# B&R Automation Studio project Soiled_PLC (part 17)

#### Main.st
```iecst
PROGRAM _INIT
	state 			:= 0;
	pFileName 	:= ADR('Test');//file name
	pFileDevice	:=ADR('FTP');//Can be file name set up in AS, or Devlink folder name
	//pDevLinkParameter := ADR('/DEVICE=C:\\Projects\FTP\Test');//Path for Devlink
	pDevLinkParameter := ADR('/SIP=10.8.4.211 /PROTOCOL=ftp /USER=SUP /PASSWORD=12345');
	pMemCard	:= ADR('memcard');//Pointer to memory card file device
	pUSB 		:= ADR('USB');
	//Create temporary memory object for the files to be read into..
	sizeTempMem := 30000000; //Allocate 30MB of free memory
	TMP_alloc(sizeTempMem,ADR(pTempMem));
END_PROGRAM

PROGRAM _CYCLIC

	CASE state OF
		XML_READER_IDLE:

		XML_READER_COPY_FILE_TO_MEMCARD: //Copy File from FTP Server to Memcard.
			fileCopyFromDev.enable := 1;
			fileCopyFromDev.pFileName := pFileName;// Name of file to copy
			fileCopyFromDev.pFileDevice := pFileDevice;//Folder to copy from
			fileCopyFromDev.pDevLinkParameter := pDevLinkParameter;//Parameters for Devlink...
			fileCopyFromDev.pDest := pFileName;
			fileCopyFromDev.pDestDev := pMemCard;//pUSB;
			fileCopyFromDev();
			IF fileCopyFromDev.status = ERR_OK THEN
				state := XML_READER_DECODE_FILE;
			ELSIF fileCopyFromDev.status = 26228 THEN//ERR_DDFI_NETIO_DLINK THEN //No file available on network... use local memory card file..
				state := XML_READER_DECODE_FILE;
			ELSIF fileCopyFromDev.status <> ERR_FUB_BUSY THEN
				state := XML_READER_DECODE_ERROR;
			END_IF;

		XML_READER_DECODE_FILE:
		//Decode XML File Copy into temp memory then read...
			n:= 0;
			FOR n:= 0 TO 100 DO //Use loop to increase scan time..
				CASE xmlReader OF
					0://Copy into memory
						fiToMem.enable := 1;
						fiToMem.pFileDevice := pMemCard;
						fiToMem.pFileName := pFileName;
						fiToMem.pTempMem := pTempMem;
						fiToMem.sizeTempMem := sizeTempMem;
						fiToMem();
						IF fiToMem.status = ERR_OK THEN
							memcpy(ADR(testString),pTempMem,SIZEOF(testString));
							xmlReader := 10;
						ELSIF fiToMem.status <> ERR_FUB_BUSY THEN
							xmlReader := 100;
						END_IF;

					10://Copy data to file for test..
						fileWrite.enable := 1;
						fileWrite.mode := FILE_SAVE;
						fileWrite.Offset := 0;
						fileWrite.pData := pTempMem;
						fileWrite.sizeData := fiToMem.fiSize;//responseHeader.contentLength;
						fileWrite.pFileDevice := pUSB;
						fileWrite.pFileName := ADR('FTP_Test.xml');
						fileWrite();
						IF fileWrite.status = ERR_OK THEN
							xmlReader := 1;
						END_IF;

					1://Create XML Reaser
						xmlReadCreate.enable := 1;
						xmlReadCreate.memorySize := fiToMem.fiSize;
						xmlReadCreate.pXmlMemory := pTempMem;
						xmlReadCreate();
						IF xmlReadCreate.status = ERR_OK THEN
							lineCount := 0;
							xmlReader := 2;
						ELSIF xmlReadCreate.status <> ERR_FUB_BUSY THEN
							xmlReader := 100;
						END_IF;

					2://Search for 'Config setting'
						xmlReadNode.enable := 1;
						xmlReadNode.ident := xmlReadCreate.ident;
						xmlReadNode.forceRead := 0;
						xmlReadNode.skipSubtree := 0;
						xmlReadNode.pName := ADR(xmlName);
						xmlReadNode.nameSize := SIZEOF(xmlName);
						xmlReadNode.pValue := ADR(xmlValue);
						xmlReadNode.valueSize := SIZEOF(xmlValue);
						xmlReadNode();
						IF xmlReadNode.status = ERR_OK THEN
							IF xmlName = 'Config' THEN
								lineCount := lineCount + 1;
								xmlIndex := 0;
								xmlReader := 3;
							END_IF;
						ELSIF xmlReadNode.status = xmlERR_NO_FURTHER_XML_NODE THEN
							xmlReader := 4;//End of file
						ELSIF xmlReadNode.status <> ERR_FUB_BUSY THEN
							xmlReader := 100;
						END_IF

					3://Decode XML elements
						xmlReadAttNum.enable := 1;
						xmlReadAttNum.ident := xmlReadCreate.ident;
						xmlReadAttNum.index := xmlIndex;
						xmlReadAttNum.pName := ADR(xmlName);
						xmlReadAttNum.nameSize := SIZEOF(xmlName);
						xmlReadAttNum.pValue := ADR(xmlValue);
						xmlReadAttNum.valueSize := SIZEOF(xmlValue);
						xmlReadAttNum();
						IF xmlReadAttNum.status = ERR_OK THEN
							IF xmlName = 'Property' THEN
								xmlProperty := xmlValue;
							ELSIF xmlName = 'Index' THEN
								xmlPropertyIndex := atoi(ADR(xmlValue));
							ELSIF xmlName =	'FirstBag' THEN
								IF (xmlProperty = 'Line') AND (xmlPropertyIndex > 0) AND  (xmlPropertyIndex <= MAX_LINES) THEN
									Line[xmlPropertyIndex].FirstBag := DINT_TO_UINT(atoi(ADR(xmlValue)));
								END_IF;
							ELSIF xmlName = 'LastBag' THEN
								IF (xmlProperty = 'Line') AND (xmlPropertyIndex > 0) AND  (xmlPropertyIndex <= MAX_LINES) THEN
									Line[xmlPropertyIndex].LastBag := DINT_TO_UINT(atoi(ADR(xmlValue)));
								END_IF;
							END_IF;
							xmlIndex := xmlIndex + 1;
						ELSIF xmlReadAttNum.status = xmlERR_INVALID_ATTRIBUTE_INDEX THEN//No more elements go back to beginning..
							xmlReader := 2;
						ELSIF xmlReadAttNum.status <> ERR_FUB_BUSY THEN
							xmlReader := 100;
						END_IF

					4://Close XML Reader
						xmlCloseReader.enable := 1;
						xmlCloseReader.ident := xmlReadCreate.ident;
						xmlCloseReader();
						IF xmlCloseReader.status = ERR_OK THEN
							xmlReader := 99;
						ELSIF xmlCloseReader.status <> ERR_FUB_BUSY THEN
							xmlReader := 100;
						END_IF;

					99:
						state := 99;
						xmlReader := 0;
					100://Error
						state := 100;
						xmlReader := 0;

				END_CASE;
				IF xmlReader = 0 THEN
					EXIT;
				END_IF;
			END_FOR;

		XML_READER_DECODE_ERROR:

		ELSE
			state := XML_READER_IDLE;

	END_CASE;

END_PROGRAM
```

### Program Logical/File_System/zzXMLFileViaHttp (IEC)

#### Variables.var
```iecst
(*State Constants*)
VAR CONSTANT
	XML_READER_IDLE : UINT := 0;
	XML_READER_READ_FROM_HTTP : UINT := 1;
	XML_READER_DECODE_FILE : UINT := 2;
	XML_READER_DECODE_ERROR : UINT := 99;
END_VAR
(**Local Vars*)
VAR
	state : UINT;
	error : UINT;
	pTempMem : UDINT;
	sizeTempMem : UDINT;
	pFileName : UDINT;
	pFileDevice : UDINT;
	pDevLinkParameter : UDINT;
	pMemCard : UDINT;
	fileCopyFromDev : FileCopyFromDev;
	pUSB : UDINT;
	n : UINT;
	xmlReader : UINT;
	lineCount : UINT;
	xmlName : STRING[100];
	xmlValue : STRING[100];
	xmlIndex : UDINT;
	xmlProperty : STRING[100];
	xmlPropertyIndex : DINT;
	fiToMem : fileToMem;
	xmlReadCreate : xmlCreateMemoryReader;
	xmlReadNode : xmlReadNextNode;
	xmlReadAttNum : xmlReadAttributeNr;
	xmlCloseReader : xmlCloseMemoryReader;
	pHost : UDINT;
	URL : STRING[30];
	pResponseHeader : UDINT;
	responseHeader : httpResponseHeader_t;
	pRequestHeader : UDINT;
	requestHeader : httpRequestHeader_t;
	pStatistics : UDINT;
	Statistics : httpStatistics_t;
	pSendData : UDINT;
	sendData : STRING[100];
	pResponseData : UDINT;
	responseData : ARRAY[0..99] OF USINT;
	pUri : UDINT;
	testAbort : BOOL;
	http_Client : httpClient;
	testSend : BOOL;
	fileWrite : fileReadWrite;
	fiLength : UDINT;
END_VAR
```

#### Main.st
```iecst
PROGRAM _INIT
	pHost := ADR('10.8.4.102');
	URL := '/plctalk/api/values/3';
	pUri := ADR(URL);
	pResponseHeader := ADR(responseHeader);
	pRequestHeader := ADR(requestHeader);
	pStatistics := ADR(Statistics);
	pSendData := ADR(sendData);
	pResponseData := ADR(responseData);

	state 			:= 0;
	pFileName 	:= ADR('Test');//file name
	//pFileDevice	:=ADR('FTP');//Can be file name set up in AS, or Devlink folder name
	//pDevLinkParameter := ADR('/DEVICE=C:\\Projects\FTP\Test');//Path for Devlink
	//pDevLinkParameter := ADR('/SIP=10.8.4.211 /PROTOCOL=ftp /USER=SUP /PASSWORD=12345');
	pMemCard	:= ADR('memcard');//Pointer to memory card file device
	pUSB 		:= ADR('USB');
	//Create temporary memory object for the files to be read into..
	sizeTempMem := 10000000; //Allocate 10MB of free memory
	TMP_alloc(sizeTempMem,ADR(pTempMem));
END_PROGRAM

PROGRAM _CYCLIC
http_Client.enable := 1;
http_Client.send := testSend;
http_Client.abort := testAbort;
http_Client.option := httpOPTION_HTTP_11;
http_Client.pHost := pHost;
http_Client.hostPort := 0;//20997;
http_Client.pUri := pUri;
http_Client.pRequestHeader := 0;//pRequestHeader;
http_Client.pRequestData := pSendData;
http_Client.requestDataLen := LEN(sendData);
http_Client.pResponseHeader := pResponseHeader;
http_Client.pResponseData := pTempMem; //pResponseData;
http_Client.responseDataSize := sizeTempMem;//SIZEOF(responseData);
http_Client.pStatistics := pStatistics;
http_Client.method := httpMETHOD_GET;
http_Client();

	CASE state OF
		XML_READER_IDLE:
			testSend := 0;

		XML_READER_READ_FROM_HTTP: //Copy File from FTP Server to Memcard.
			testSend := 1;
			IF (http_Client.phase = httpPHASE_RECEIVED) THEN
				state := 10;//XML_READER_DECODE_FILE;
				IF (responseHeader.contentLength > 0) THEN
					IF (responseHeader.contentLength <= SIZEOF(responseData)) THEN
						memcpy(pResponseData,pTempMem,responseHeader.contentLength);
					ELSE
						memcpy(pResponseData,pTempMem,SIZEOF(responseData));
					END_IF;
				END_IF;
			END_IF;

		10://Copy data to file for test..
			fileWrite.enable := 1;
			fileWrite.mode := FILE_SAVE;
			fileWrite.Offset := 0;
			fileWrite.pData := pTempMem;
			fileWrite.sizeData := responseHeader.contentLength;
			fileWrite.pFileDevice := pUSB;
			fileWrite.pFileName := ADR('text.xml');
			fileWrite();
			IF fileWrite.status = ERR_OK THEN
				state := XML_READER_DECODE_FILE;
			ELSIF fileWrite.status <> ERR_FUB_BUSY THEN
				state := XML_READER_DECODE_FILE;
			END_IF;

		XML_READER_DECODE_FILE:
		//Decode XML File Copy into temp memory then read...
			n:= 0;
			FOR n:= 0 TO 100 DO //Use loop to increase scan time..
				CASE xmlReader OF
					0://Copy into memory
//						fiToMem.enable := 1;
//						fiToMem.pFileDevice := pMemCard;
//						fiToMem.pFileName := pFileName;
//						fiToMem.pTempMem := pTempMem;
//						fiToMem.sizeTempMem := sizeTempMem;
//						fiToMem();
//						IF fiToMem.status = ERR_OK THEN
							xmlReader := 1;
//						ELSIF fiToMem.status <> ERR_FUB_BUSY THEN
//							xmlReader := 100;
//						END_IF;

					1://Create XML Reaser
						xmlReadCreate.enable := 1;
						xmlReadCreate.memorySize := responseHeader.contentLength;
						xmlReadCreate.pXmlMemory := pTempMem;
						xmlReadCreate();
						IF xmlReadCreate.status = ERR_OK THEN
							lineCount := 0;
							xmlReader := 2;
						ELSIF xmlReadCreate.status <> ERR_FUB_BUSY THEN
							xmlReader := 100;
						END_IF;

					2://Search for 'Config setting'
						xmlReadNode.enable := 1;
						xmlReadNode.ident := xmlReadCreate.ident;
						xmlReadNode.forceRead := 0;
						xmlReadNode.skipSubtree := 0;
						xmlReadNode.pName := ADR(xmlName);
						xmlReadNode.nameSize := SIZEOF(xmlName);
						xmlReadNode.pValue := ADR(xmlValue);
						xmlReadNode.valueSize := SIZEOF(xmlValue);
						xmlReadNode();
						IF xmlReadNode.status = ERR_OK THEN
							IF xmlName = 'Config' THEN
								lineCount := lineCount + 1;
								xmlIndex := 0;
								xmlReader := 3;
							END_IF;
						ELSIF xmlReadNode.status = xmlERR_NO_FURTHER_XML_NODE THEN
							xmlReader := 4;//End of file
						ELSIF xmlReadNode.status <> ERR_FUB_BUSY THEN
							xmlReader := 100;
						END_IF

					3://Decode XML elements
						xmlReadAttNum.enable := 1;
						xmlReadAttNum.ident := xmlReadCreate.ident;
						xmlReadAttNum.index := xmlIndex;
						xmlReadAttNum.pName := ADR(xmlName);
						xmlReadAttNum.nameSize := SIZEOF(xmlName);
						xmlReadAttNum.pValue := ADR(xmlValue);
						xmlReadAttNum.valueSize := SIZEOF(xmlValue);
						xmlReadAttNum();
						IF xmlReadAttNum.status = ERR_OK THEN
							IF xmlName = 'Property' THEN
								xmlProperty := xmlValue;
							ELSIF xmlName = 'Index' THEN
								xmlPropertyIndex := atoi(ADR(xmlValue));
							ELSIF xmlName =	'FirstBag' THEN
								IF (xmlProperty = 'Line') AND (xmlPropertyIndex > 0) AND  (xmlPropertyIndex <= MAX_LINES) THEN
									Line[xmlPropertyIndex].FirstBag := DINT_TO_UINT(atoi(ADR(xmlValue)));
								END_IF;
							ELSIF xmlName = 'LastBag' THEN
								IF (xmlProperty = 'Line') AND (xmlPropertyIndex > 0) AND  (xmlPropertyIndex <= MAX_LINES) THEN
									Line[xmlPropertyIndex].LastBag := DINT_TO_UINT(atoi(ADR(xmlValue)));
								END_IF;
							END_IF;
							xmlIndex := xmlIndex + 1;
						ELSIF xmlReadAttNum.status = xmlERR_INVALID_ATTRIBUTE_INDEX THEN//No more elements go back to beginning..
							xmlReader := 2;
						ELSIF xmlReadAttNum.status <> ERR_FUB_BUSY THEN
							xmlReader := 100;
						END_IF

					4://Close XML Reader
						xmlCloseReader.enable := 1;
						xmlCloseReader.ident := xmlReadCreate.ident;
						xmlCloseReader();
						IF xmlCloseReader.status = ERR_OK THEN
							xmlReader := 99;
						ELSIF xmlCloseReader.status <> ERR_FUB_BUSY THEN
							xmlReader := 100;
						END_IF;

					99:
						state := 99;
						xmlReader := 0;

					100://Error
						state := 100;
						xmlReader := 0;

				END_CASE;
				IF xmlReader = 0 THEN
					//memset(pTempMem,0,sizeTempMem); //Clear memory when finish
					EXIT;
				END_IF;
			END_FOR;

		XML_READER_DECODE_ERROR:

		100://ERROR

		ELSE
			state := XML_READER_IDLE;

	END_CASE;

END_PROGRAM
```

### Program Logical/File_System/sendXML (IEC)

#### Variables.var - Local variables
```iecst
VAR
	xml : xml_typ;
	state : REFERENCE TO USINT;
	xmlWriter : xml_writer_typ;
	testData : testData_typ;
	status : UINT;
	pStructName : UDINT;
	index : UINT;
	pvName : STRING[50];
	structName : STRING[32];
	taskName : STRING[55];
	encodeXML : WriteXMLFromStructure;
	pv_dataLen : UINT;
	noOfElements : UINT;
	pvStatus : UINT;
	pv_dataType : UINT;
	pvFullName : STRING[50];
	subIndex : UINT;
	pvValue : UDINT;
	batch : test2;
	enable : BOOL;
	testTim : BOOL;
END_VAR
```

#### Types.typ - Local data types
```iecst
TYPE
	xml_typ : 	STRUCT
		Write : xml_writer_typ;
	END_STRUCT;
	xml_writer_typ : 	STRUCT
		State : USINT; (**State of the writer...*)
		Functions : xml_write_fub_typ;
	END_STRUCT;
	xml_write_fub_typ : 	STRUCT
		CreateMemWriter : xmlCreateMemoryWriter;
	END_STRUCT;
	testData_typ : 	STRUCT
		BatchID : USINT;
		ElementArray : ARRAY[0..9]OF USINT;
		Structure : test2;
	END_STRUCT;
	test2 : 	STRUCT
		StrElement : USINT;
		stElement2 : USINT;
	END_STRUCT;
END_TYPE
```

#### Main.st - Init, cyclic, exit code
```iecst
PROGRAM _INIT
	(* Insert code here *)

END_PROGRAM

PROGRAM _CYCLIC
	//_compileXML;
	DF2327SortedBatches;

	DF2327SortedBatches.updatedAt := CurrentTimestamp;
	batch;

	encodeXML.enable := enable;
	encodeXML.pStructName := ADR('DF2327SortedBatches');
	encodeXML.pData := ADR(Data);
	encodeXML.sizeData := SIZEOF(Data);
	encodeXML();
	IF (encodeXML.status = ERR_OK) THEN
		enable := 0;
	ELSIF (encodeXML.status <> ERR_FUB_BUSY) THEN

	END_IF;

	IF testTim THEN
		memcpy(ADR(Data),ADR(''),SIZEOF(Data));
		testTim := 0;
	 END_IF;
END_PROGRAM
```

#### compileXML.st
```iecst
ACTION _compileXML:
	state ACCESS ADR(xml.Write.State);
	testData;

	CASE xmlWriter.State OF

		30://Open an XML writer
			xmlWriter.Functions.CreateMemWriter.enable := 1;
			IF (xmlWriter.Functions.CreateMemWriter.status = ERR_OK) THEN
				xmlWriter.State := 1;
			END_IF;

		1:// Write the document header
			//Write the encoding version.

		10://Wait.
			structName := 'testData';
			pStructName := ADR(structName);

		11://Read the Data structure so we can manipulate into XML
			//What have to pass in the structure Name..
			// Only pass the structure name -- The code will handle it if it;s global or local
			status := PV_item(pStructName,index,ADR(pvName));
			IF (status = ERR_OK) THEN
				//Build the pvFullName
				brsstrcpy(ADR(pvFullName),ADR(structName));
				brsstrcat(ADR(pvFullName),ADR('.'));
				brsstrcat(ADR(pvFullName),ADR(pvName));
				xmlWriter.State := 20;
			ELSIF (status =  ERR_SYS_PV_NOT_FOUND) THEN
				//Add the taskname in front of the var to declare it as local.
				ST_name(0,ADR(taskName),0);
				brsstrcat(ADR(taskName),ADR(':'));
				brsstrcat(ADR(taskName),ADR(structName));
				brsstrcpy(ADR(structName),ADR(taskName));
				pStructName := ADR(structName);
			END_IF;

		20://Get the info..
			pvStatus := PV_ninfo(ADR(pvFullName),ADR(pv_dataType),ADR(pv_dataLen),ADR(noOfElements));
			IF pvStatus = ERR_OK THEN
				xmlWriter.State := 21;
			END_IF;

		21://
			//Don't use get val as it doesn;t support strings..
			//We can get the address and memcpy... then cast to string

			//pvStatus := PV_xgetval(ADR(pvFullName),subIndex,ADR(pvValue),2);
			IF pvStatus = ERR_OK THEN
				xmlWriter.State := 22;
			END_IF;

		99://Close the writer.
			//xml

	END_CASE;

END_ACTION
```

### Program Logical/ExportsFromOriginal/0_sbelt (IEC, version 1.00.0) - * Loading and Sorting belts

#### 0_sbeltCyclic.ab
```automation-basic
PROGRAM _CYCLIC
(* cyclic program *)

;Inputs
I_SortBelt3Photo	= X[3].X16

O_RunSortBelt1 		= FALSE
O_RunSortBelt2 		= FALSE
O_RunSortBelt3 		= FALSE

;Run belts
O_RunSortBelt3 = NOT I_SortBelt3Photo AND NOT Std.EStopLoading ;Std.EStop
TON_10ms(O_RunSortBelt3,300,O_RunSortBelt2,SortBelt3RunningET)
TON_10ms(O_RunSortBelt2,300,O_RunSortBelt1,SortBelt2RunningET)

;Outputs
Y[2].Y11 = O_RunSortBelt3
;Y[13].Y09 = O_RunSortBelt2
;Y[13].Y11 = O_RunSortBelt3

END_PROGRAM
```

#### 0_sbelt.var
```iecst
VAR
	I_SortBelt3Photo	:BOOL;
	O_RunSortBelt1	:BOOL;
	O_RunSortBelt2	:BOOL;
	O_RunSortBelt3	:BOOL;
	SortBelt2RunningET	:TIME;
	SortBelt3RunningET	:TIME;
END_VAR
```

### Program Logical/ExportsFromOriginal/1_stnsa (IEC, version 1.00.0) - * Honeycombe Stations 1 - 16

#### 1_stnsaCyclic.ab
```automation-basic
PROGRAM _CYCLIC
	(* cyclic program *)

;Honeycombe Sorting Station Control
;----------------------------------------------------
;Revision 1.00 10/01/2002 D.J. First Issue
;Revision 2.00 07/02/2005 D.J. Removed Stn Mix
;Revision 3.00 22/08/2006 D.J. Changed to timer array
;----------------------------------------------------

Bank = 1

;Timers
OpenTime  = 700
CloseTime = 300

LOOP n = Ldg[Bank].StartStn TO Ldg[Bank].EndStn DO

	;Bag open timers
	TimerOpen[n].IN 	= OpenBag[n]
	TimerOpen[n].PT		= OpenTime
	TimerOpen[n] FUB TON_10ms()

	BagOpened[n] 		= TimerOpen[n].Q
	BagOpenedET[n]		= TimerOpen[n].ET

	;Bag closed timers
	TimerClosed[n].IN 	= NOT OpenBag[n]
	TimerClosed[n].PT	= CloseTime
	TimerClosed[n] FUB TON_10ms()

	BagClosed[n] 		= TimerClosed[n].Q
	BagClosedET[n]		= TimerClosed[n].ET

	;Update bag weight
	StnBag = n + (Std.StationBagsStart[Bank] - 1)
	Bag[StnBag].Wgt = Stn[n].Weight
	Bag[StnBag].Cnt = Stn[n].Count

	Alarm[40 + n].Name 		= 0
	Alarm[40 + n].Bag		= StnBag
	Alarm[40 + n].Beacon	= TRUE
	Alarm[40 + n].Extra		= 0
	Alarm[40 + n].Time		= 2000

	Stn[n].LampOn 		= FALSE

	STEP = D[940 + n]
	;Setup Pulse contact
	PLS[n] = (STEP <> LASTSTEP[n])
	LASTSTEP[n] = STEP

	;Step 0 - Disabled
	IF (STEP = 0) THEN
		Stn[n].LampOn = TRUE
		;Disabled
	ENDIF

	IF (STEP = 1) THEN
		Stn[n].LampOn = TRUE
		IF D[901] = n THEN
			D[901] = 0
		ENDIF
		IF BagClosed[n] THEN
			D[940 + n] = 2
		ENDIF
		Alarm[40 + n].Name = almStationNotClosed
	ENDIF

	IF (STEP = 2) THEN
		Stn[n].LampOn = ((Stn[n].SP1 AND Std.Clock2s) OR Stn[n].SP2 OR (Stn[n].SP3 AND Std.Clock200ms))
		IF ((D[901] = n) AND Ldg[Bank].EnableStnRelease) THEN
			D[940 + n] = 3
		ENDIF
		IF ((Bag[StnBag].Cat > 0) AND Stn[n].SP3) THEN
			Alarm[40 + n].Name = almBagOverWeight
		ENDIF
	ENDIF

	IF (STEP = 3) THEN
		Stn[n].LampOn = TRUE
		IF (BagOpened[n] AND ((Stn[n].Weight < 30) OR Test.Stations) AND Ldg[Bank].BeltHasRun) THEN
			Stn[n].QTime 	= 0
			D[940 + n] 		= 1
		ENDIF
		IF (Stn[n].Weight >= 30) THEN
			Alarm[40 + n].Name = almStationNotEmpty
		ENDIF
	ENDIF

	OpenBag[n] = (STEP = 3)

	;Alarm timer
	TimerAlarm[n].IN 	= NOT PLS[n] AND (Alarm[40 + n].Name > 0)
	TimerAlarm[n].PT	= Alarm[40 + n].Time
	TimerAlarm[n] FUB TON_10ms()

	Alarm[40 + n].ET	= TimerAlarm[n].ET
	Alarm[40 + n].On 	= TimerAlarm[n].Q

ENDLOOP

;Outputs
;-------

Y[31].Y05 = OpenBag[1]
Y[31].Y06 = OpenBag[2]
Y[31].Y07 = OpenBag[3]
Y[31].Y08 = OpenBag[4]
Y[31].Y13 = OpenBag[5]
Y[31].Y14 = OpenBag[6]
Y[31].Y15 = OpenBag[7]
Y[31].Y16 = OpenBag[8]
Y[32].Y05 = OpenBag[9]
Y[32].Y06 = OpenBag[10]
Y[32].Y07 = OpenBag[11]
Y[32].Y08 = OpenBag[12]
Y[32].Y13 = OpenBag[13]
Y[32].Y14 = OpenBag[14]
Y[32].Y15 = OpenBag[15]
Y[32].Y16 = OpenBag[16]

Y[31].Y01 = Stn[1].LampOn
Y[31].Y02 = Stn[2].LampOn
Y[31].Y03 = Stn[3].LampOn
Y[31].Y04 = Stn[4].LampOn
Y[31].Y09 = Stn[5].LampOn
Y[31].Y10 = Stn[6].LampOn
Y[31].Y11 = Stn[7].LampOn
Y[31].Y12 = Stn[8].LampOn
Y[32].Y01 = Stn[9].LampOn
Y[32].Y02 = Stn[10].LampOn
Y[32].Y03 = Stn[11].LampOn
Y[32].Y04 = Stn[12].LampOn
Y[32].Y09 = Stn[13].LampOn
Y[32].Y10 = Stn[14].LampOn
Y[32].Y11 = Stn[15].LampOn
Y[32].Y12 = Stn[16].LampOn
END_PROGRAM
```

#### 1_stnsa.var
```iecst
VAR RETAIN
	n	:UINT;
	OpenBag	:ARRAY [0..99] OF BOOL;
	STEP	:UINT;
	PLS	:ARRAY [0..99] OF BOOL;
	LASTSTEP	:ARRAY [0..99] OF UINT;
	BagClosed	:ARRAY [0..99] OF BOOL;
	BagClosedET	:ARRAY [0..99] OF TIME;
	OpenTime	:UINT;
	BagOpenedET	:ARRAY [0..99] OF TIME;
	BagOpened	:ARRAY [0..99] OF BOOL;
	CloseTime	:UINT;
END_VAR

VAR
	Bank	:UINT;
	TimerOpen	:ARRAY [0..49] OF TON_10ms;
	TimerClosed	:ARRAY [0..49] OF TON_10ms;
	TimerAlarm	:ARRAY [0..49] OF TON_10ms;
	StnBag	:UINT;
END_VAR
```

### Program Logical/ExportsFromOriginal/2_belt1 (IEC, version 2.00.0) - * Transfer Belt 1

#### 2_belt1Cyclic.ab
```automation-basic
PROGRAM _CYCLIC
 	(* cyclic program *)

;Sequence 2 - Transfer Belt 1 from Stations 1-12

;-----------------------------------------
;Revision 1.00 18/01/2006 D.J. First Issue
;-----------------------------------------

;Inputs and Outputs
;------------------

Bank 						= 1

I_PhotoBottom 				= X[3].X08
I_PhotoTop   				= X[3].X08

Request.TransferBelt[Bank]	= FALSE

O_RunBelt 					= FALSE

Alarm[2].Name 				= 0
Alarm[2].Bag				= 220
Alarm[2].Beacon				= TRUE
Alarm[2].Extra				= 0
Alarm[2].Time				= 5000

n = D[901] ;Selected Station

STEP = D[902]
;Setup Pulse contact
PLS = (STEP <> LASTSTEP)
LASTSTEP = STEP

;Step 0 - Disabled
IF STEP = 0 THEN
	;Disabled
ENDIF

;Step 1 - Check no stations are releasing
IF STEP = 1 THEN
	;Don't allow stations to release
	Ldg[Bank].EnableStnRelease = FALSE
	;No Station Releaseng and switched on
	IF ((D[901] = 0) AND (D[11] > 0)) THEN
		IF (Bag[220].Cat = 0) THEN
			D[902] = 2 ;No Bag on belt
		ELSE
			D[902] = 4 ;Bag on belt
		ENDIF
	ENDIF
	Alarm[2].Name = almNoAlarm
ENDIF

;Step 2 - Enable Station search
IF STEP = 2 THEN

	;Check each station to see if a manual destination has been set
	LOOP n = Ldg[Bank].StartStn TO Ldg[Bank].EndStn DO

		StnBag = n + (Std.StationBagsStart[Bank] - 1)

		IF ((Bag[StnBag].Dst > 0) AND (Bag[StnBag].Dst < 99) AND (D[11] > 0)) THEN ;Dest 99 = Empty Bag in station
			Stn[n].DestManual = Bag[StnBag].Dst
		ELSE
			Stn[n].DestManual = 0
		ENDIF
		;For pairing set number of spaces to search for
		Stn[n].SpacesRequired = 0 ;D[2000 + Bag[StnBag].Cat]

	ENDLOOP

	;Station Search
	IF ((Ldg[Bank].Search = 0) AND (D[11] > 0) AND NOT Std.EStop) THEN
		Ldg[Bank].Search = 1
	ELSE IF ((Ldg[Bank].Search = 2) AND (Ldg[Bank].Found > 0))  THEN

		D[901] 	= Ldg[Bank].Found
		n 		= D[901]

		StnBag 	= n + (Std.StationBagsStart[Bank] - 1)

		;Clear the release button count if used
		Stn[n].ManualRelease 	= FALSE
		Stn[n].PBCount 			= 0

		;------Write Report------
		IF Std.StationReports  THEN

			IF (ReportLoading[n].Cat = 0) THEN

				;Check if anything has been added and current weight is not less than the previous
				WeightValue = Stn[n].Weight - INT(StnPrev[n].Wgt)
				WeightValid = (WeightValue > 0)

				IF WeightValid THEN

					;Ensure valid values as we report on either a weight or count change
					IF (WeightValue < 0) THEN
						WeightValue = 0
					ENDIF

					ReportLoading[n].Cat = UINT(Bag[StnBag].Cat)	;Category
					ReportLoading[n].Cus = Bag[StnBag].Cus			;Customer
					ReportLoading[n].Wgt = UINT(WeightValue)		;Weight
					ReportLoading[n].Cnt = 0						;Count
					ReportLoading[n].Stn = n         				;Station
					ReportLoading[n].Mcn = 0						;Machine

				ENDIF

			ENDIF

		ENDIF

		;Set Previous Cat and Cus to Current and Clear Weight and Count
		StnPrev[n].Cat 	= Bag[StnBag].Cat
		StnPrev[n].Cus 	= Bag[StnBag].Cus
		StnPrev[n].Wgt 	= 0

		;Copy Station Data to Belt Bag
		Bag[220] 		= Bag[StnBag]			;Copy complete bag data
		Bag[220].Dst 	= USINT(Ldg[Bank].Line)	;Destination
		Bag[StnBag].Dst = 0 					;Reset Destination (Manual)

		;Clear Manual Release
		Stn[n].ManualRelease = FALSE

		;If Stations are too close to the loading unit then jump to wait for loading unit
		;IF (n >= 1) AND (n <= 4) THEN
		;	D[902] = 6
		;ELSE
			BeltAddTime = (D[901] / 2)
			Ldg[Bank].EnableStnRelease = TRUE
			D[902] = 3
		;ENDIF

		Alarm[2].Name = almNoAlarm

	ENDIF
ELSE
	Ldg[Bank].Search  	= 0 ;Clear Search if not on step 2
ENDIF

;Step 3
;Open Bag and Release to Belt Conveyor
IF STEP = 3 THEN
;	O_RunBelt  = TRUE
;	IF (I_PhotoBottom OR I_PhotoTop	OR Test.TransferBelt) THEN
		D[902] = 4
;	ENDIF
;	Alarm[2].Name = almPhotocellNotMade
ENDIF

;Step 4 - Skipped
IF STEP = 4 THEN
	O_RunBelt = TRUE
	D[902] = 5
	Alarm[2].Name = almNoAlarm
ENDIF

;Step 5 - Run belt until top photocell is made.
IF STEP = 5 THEN
	O_RunBelt = TRUE
	IF I_PhotoTop OR Test.TransferBelt THEN
		D[902] = 6
	ENDIF
	Alarm[2].Name = almPhotocellNotMade
ENDIF

;Step 6 - Wait for loading unit ready
TON_10ms((STEP = 6),10,RunBelt,Step6ET)
IF STEP = 6 THEN
	O_RunBelt = (NOT RunBelt AND Ldg[Bank].EnableStnRelease)
	IF Enable.TransferBelt[Bank] THEN
		D[902] = 7
	ENDIF
ENDIF

;Step 7 - Run Belt until linen detected for 1 second and Station has emptied
TON_10ms(((STEP = 7) AND I_PhotoTop),100,LinenDetected,LinenDetectedET)
IF STEP = 7 THEN
	O_RunBelt = TRUE
	Ldg[Bank].EnableStnRelease = TRUE ;Enable Station to Open bags if they haven't been already
	IF (LinenDetected OR Test.TransferBelt) THEN
		D[902] = 8
	ENDIF
	Alarm[2].Name = almPhotocellNotMade
ENDIF

;Step 8 - Run Belt until photocells clear for 5 seconds
;TON_10ms(((STEP = 8) AND NOT I_PhotoBottom AND NOT I_PhotoTop AND NOT Std.EStop),500,BeltClear,BeltClearET)
TON_10ms(((STEP = 8) AND NOT I_PhotoBottom AND NOT I_PhotoTop AND NOT Std.EStopLoading),500,BeltClear,BeltClearET)
IF STEP = 8 THEN
	O_RunBelt = TRUE
	IF (BeltClear AND MinBeltRun AND (D[901] = 0)) THEN
		D[902] = 9
	ENDIF
	IF NOT Std.EStopLoading THEN
		IF I_PhotoBottom OR I_PhotoTop THEN
			Alarm[2].Name = almPhotocellBlocked
		ELSE IF (D[901] <> 0) THEN
			Alarm[2].Name = almStationNotClosed
		ELSE IF NOT MinBeltRun THEN
			Alarm[2].Name = almClearingBeltPleaseWait
		ENDIF
	ENDIF
ENDIF

;Note - Unitl the Station has closed the min belt run time won't start
BeltRunTime = (12 + BeltAddTime)
CTU((O_RunBelt AND Std.Clock1s AND (D[901] = 0) AND NOT Std.EStop),(STEP = 1),BeltRunTime,MinBeltRun,MinBeltRunCV)

;Step 9 - Check Stations Are Closed
IF STEP = 9 THEN
	;Move Belt bag to loading unit
	IF PLS AND (Bag[221].Cat = 0) AND (Bag[220].Cat > 0) THEN
		Bag[221] = Bag[220]
		Bag[220] = Bag[0]
	ENDIF
	IF (D[901] = 0) THEN
		D[902] = 1
	ENDIF
	Alarm[2].Name = almStationNotClosed
ENDIF

;Alarms
TimerAlarm.IN = NOT PLS AND (Alarm[2].Name > 0)
TimerAlarm.PT = Alarm[2].Time
TimerAlarm FUB TON_10ms()
Alarm[2].On = TimerAlarm.Q
Alarm[2].ET = TimerAlarm.ET

;Outputs
;Inform Station Sequences that the belt has been
Ldg[Bank].BeltHasRun = ((D[902] > 3) AND Ldg[Bank].EnableStnRelease)

Y[2].Y10 = O_RunBelt
END_PROGRAM
```

#### 2_belt1.var
```iecst
VAR RETAIN
	MinBeltRunCV	:UINT;
	MinBeltRun	:BOOL;
	BeltClearET	:TIME;
	BeltClear	:BOOL;
	LinenDetectedET	:TIME;
	LinenDetected	:BOOL;
	n	:UINT;
	STEP	:UINT;
	Step6ET	:TIME;
	LASTSTEP	:UINT;
	PLS	:BOOL;
	O_RunBelt	:BOOL;
	RunBelt	:BOOL;
END_VAR

VAR
	TimerAlarm	:TON_10ms;
	I_PhotoBottom	:BOOL;
	I_PhotoTop	:BOOL;
	Bank	:UINT;
	WeightValid	:BOOL;
	WeightValue	:INT;
	BeltRunTime	:UINT;
	BeltAddTime	:UINT;
	StnBag	:UINT;
END_VAR
```

### Program Logical/ExportsFromOriginal/3_slu_1 (IEC, version 1.00.0) - * Loading unit SLU1

#### 3_slu_1Cyclic.ab
```automation-basic
PROGRAM _CYCLIC
	(* cyclic program *)

;--------------------------------
;Sequence 3 - Loading Unit D[903]
;--------------------------------

;Inputs / Ouputs

Enable.TransferBelt[1]	= FALSE

I_BagAtBuffer			= FALSE ;X[12].X01
I_BagFrontPast			= X[3].X06
I_BagInLoadingUnit		= X[3].X05

I_ChuteBlocked			= X[3].X07
I_CompressorAtTop		= X[5].X13
I_CompressorAtMid		= X[5].X15
I_CompressorAtBot		= X[5].X14

O_MoveCompressorUp		= FALSE
O_MoveCompressorDn		= FALSE

I_BagAtSVC1Buffer		= FALSE ;X[12].X11
O_SVC1BufferOpen		= FALSE ;Y[12].Y11

O_OpenBufferStop		= FALSE
O_SteadyCylinders		= FALSE
O_OpenStop	 			= FALSE

Enable.SLU[1]			= FALSE

Alarm[3].Name 			= 0
Alarm[3].Bag			= 221
Alarm[3].Beacon			= TRUE
Alarm[3].Extra			= 0
Alarm[3].Time			= 3000

;Setup Sequence
;--------------
STEP = D[903]
;Setup Pulse contact
PLS = (STEP <> LASTSTEP)
LASTSTEP = STEP

IF (STEP = 0) THEN
	;Disabled
ENDIF

;Wait for Empty bag at buffer
SwitchFault = ((STEP = 1) AND (I_BagFrontPast OR I_BagInLoadingUnit))
TON_10ms(NOT SwitchFault,200,LoadingUnitClear,LoadingUnitClearET)
TON_10ms(I_BagAtBuffer,300,BagSettledBuffer,BagSettledBufferET)
IF (STEP = 1) THEN
	;IF BagSettledBuffer AND LoadingUnitClear AND NOT Std.HaltSys THEN
	IF LoadingUnitClear AND NOT Std.HaltSys THEN
		D[903] = 2
	ENDIF
	IF SwitchFault THEN
		Alarm[3].Name = almSwitchFault
	ELSE
		Alarm[3].Name = almNoAlarm
	ENDIF
ENDIF

;Open stops let bag in Loading Unit
IF (STEP = 2) THEN
	O_OpenStop 			= TRUE
	O_OpenBufferStop 	= TRUE
	Enable.SLU[1]		= NOT I_BagFrontPast
	IF I_BagFrontPast THEN
		D[903] = 3
	ENDIF
	;Alarm[3].Name = almBagNotArrived
ENDIF

;Wait for bag to settle
TON_10ms(I_BagInLoadingUnit,300,EBagSettled,EBagSettledET)
IF (STEP = 3) THEN
	IF EBagSettled THEN
		D[903] = 4
	ENDIF
	Alarm[3].Name = almBagNotSettled
	;Special for Banbury - SVC1 is also a loading hoist
	IF SVC1RequestEmpty THEN
		Bag[221].Cat 	= 99
		D[903] 			= 9
	ENDIF
ENDIF

;Steady cylinders on from steps 4 - 5
O_SteadyCylinders = ((STEP = 4) OR (STEP = 5))

;Move Steady Cylinders down
TON_10ms((STEP = 4),300,SteadysDown,SteadysDownET)
IF (STEP = 4) THEN
	IF (SteadysDown AND (Bag[221].Cat = 0)) THEN
		D[903] = 5
	ENDIF
	IF (Bag[221].Cat <> 0) THEN
		Alarm[3].Name = almBagDataError
	ELSE
		Alarm[3].Name = almNoAlarm
	ENDIF
ENDIF

;Wait for bag to be loaded
IF (STEP = 5) THEN
	Enable.TransferBelt[1] = TRUE
	IF (Bag[221].Cat > 0) THEN
		D[903] = 6
	ENDIF
	Alarm[3].Name = almNoAlarm ;Transfer belt should alarm
ENDIF

;Allow Steady Cylinders to move up
TON_10ms((STEP = 6),300,SteadysUp,SteadysUpET)
IF (STEP = 6) THEN
	IF SteadysUp THEN
		IF I_ChuteBlocked THEN
			D[903] = 7
		ELSE
			D[903] = 9
		ENDIF
	ENDIF
	Alarm[3].Name = almNoAlarm
ENDIF

;Move compressor down
IF (STEP = 7) THEN
	O_MoveCompressorDn = TRUE
	IF I_CompressorAtBot THEN
		CompressCount = CompressCount + 1
		D[903] = 8
	ENDIF
	Alarm[3].Name = almSwitchFault
ENDIF

;Move compressor up
IF (STEP = 8) THEN
	IF (I_CompressorAtMid OR I_CompressorAtTop) THEN
		IF (NOT I_ChuteBlocked OR (CompressCount >= 5)) THEN
			D[903] = 9
		ELSE IF (CompressCount < 5) THEN
			D[903] = 7 ;ReTry
		;ELSE
		;	Alarm[3].Name = almPhotocellBlocked
		;	Alarm[3].Time = 100
		ENDIF
	ELSE
		Alarm[3].Name = almSwitchFault
	ENDIF
ENDIF

;Reset Compression Counter
IF ((STEP <> 7) AND (STEP <> 8)) THEN
	CompressCount = 0
ENDIF

;Check for space at Buffer
IF (STEP = 9) THEN
	IF NOT Std.HaltSys THEN
		;IF (Bag[222].Cat = 0) AND NOT I_BagAtSVC1Buffer AND NOT O_SVC1BufferOpen THEN
		IF Enable.SVC[1] THEN
			;IF Line[16].Clear THEN
				D[903] 	= 10
			;ELSE
			;	Alarm[3].Name = almSwitchFault
			;ENDIF
		ENDIF
	ENDIF
ENDIF

;Open stop - Unitl bag out
IF (STEP = 10) THEN
	O_OpenStop = TRUE
	;IF PLS THEN
	;	C[16] = 0
	;ENDIF
	;IF Line[16].Trip THEN
	IF NOT Enable.SVC[1] THEN
		Bag[222] 	= Bag[221]
		Bag[221] 	= Bag[0]
		D[903] 		= 1
	ENDIF
	Alarm[3].Name = almBagNotReleased
ENDIF

;Alarms
TimerAlarm.IN = NOT PLS AND (Alarm[3].Name > 0)
TimerAlarm.PT = Alarm[3].Time
TimerAlarm FUB TON_10ms()
Alarm[3].On = TimerAlarm.Q
Alarm[3].ET = TimerAlarm.ET

;Outputs
;-------

;Y[12].Y01 	= O_OpenBufferStop
Y[3].Y06 	= O_SteadyCylinders
Y[3].Y05 	= O_OpenStop

Y[3].Y07 	= O_MoveCompressorDn
O_MoveCompressorUp = NOT O_MoveCompressorDn
Y[3].Y08 = O_MoveCompressorUp
END_PROGRAM
```

#### 3_slu_1.var
```iecst
VAR RETAIN
	STEP	:UINT;
	PLS	:BOOL;
	LASTSTEP	:UINT;
	EBagSettled	:BOOL;
	EBagSettledET	:TIME;
	O_OpenStop	:BOOL;
	O_SteadyCylinders	:BOOL;
	LoadingUnitClear	:BOOL;
	LoadingUnitClearET	:TIME;
END_VAR

VAR
	CompressCount	:UINT;
	O_MoveCompressorUp	:BOOL;
	SteadysUpET	:TIME;
	SteadysUp	:BOOL;
	SteadysDown	:BOOL;
	SteadysDownET	:TIME;
	I_BagAtBuffer	:BOOL;
	O_OpenBufferStop	:BOOL;
	I_BagInLoadingUnit	:BOOL;
	I_BagFrontPast	:BOOL;
	SwitchFault	:BOOL;
	TimerAlarm	:TON_10ms;
	I_CompressorAtTop	:BOOL;
	I_CompressorAtBot	:BOOL;
	I_CompressorAtMid	:BOOL;
	O_MoveCompressorDn	:BOOL;
	BagSettledBuffer	:BOOL;
	BagSettledBufferET	:TIME;
	I_BagAtSVC1Buffer	:BOOL;
	O_SVC1BufferOpen	:BOOL;
	I_ChuteBlocked	:BOOL;
END_VAR
```

### Program Logical/ExportsFromOriginal/4_spn1 (IEC) - * Soiled Ongoing Transfer Lines 1 - 14

#### 4_spn1.var
```iecst
VAR RETAIN
	n	:UINT;
	STEP	:UINT;
	ResetPointsET	:TIME;
	ResetPoints	:BOOL;
	LASTSTEP	:UINT;
	PLS	:BOOL;
	LineSelect	:ARRAY [0..19] OF BOOL;
	OnGoingEnable	:BOOL;
	O_Reset	:BOOL;
	I_BagatBuffer	:ARRAY [0..4] OF BOOL;
END_VAR

VAR
	SettledBuffer	:ARRAY [0..4] OF BOOL;
	Buffer	:UINT;
	AlarmOld	:UINT;
	BufferBag	:UINT;
	DestValid	:BOOL;
	Dest	:UINT;
	BufferDst	:UINT;
	BufferBagNum	:ARRAY [0..4] OF UINT;
	TestBuffer	:UINT;
	TimerAlarm	:TON_10ms;
	Bfr	:UINT;
	BufferSettled	:BOOL;
	BufferCat	:UINT;
	MaxBuffers	:UINT;
	Buff	:UINT;
	O_OpenSelect	:ARRAY [0..4] OF BOOL;
END_VAR
```

#### 4_spn1Cyclic.ab
```automation-basic
PROGRAM _CYCLIC
; 	(* cyclic program *)

;Sequence 4 - Ongoing To Storage D[904]

;-----------------------------------------
;Revision 1.00 09/12/2005 D.J. First Issue
;-----------------------------------------

;Inputs
OnGoingEnable 		= ((D[14] > 0) AND NOT Std.HaltSys)

I_BagatBuffer[1]	= Request.SVC[1] ;X[7].X13
;I_BagatBuffer[2]	= FALSE
;I_BagatBuffer[3]	= FALSE
;I_BagatBuffer[4]	= FALSE

O_Reset 		  	= FALSE
O_OpenSelect[1]		= FALSE
;O_OpenSelect[2]	= FALSE
;O_OpenSelect[3]	= FALSE
;O_OpenSelect[4]	= FALSE

Enable.SPN[1]		= FALSE

Alarm[4].Name 		= 0
Alarm[4].Bag		= 224
Alarm[4].Beacon		= TRUE
Alarm[4].Extra	 	= 0
Alarm[4].Time		= 3000

;Setup Sequence
;--------------
STEP = D[904]
;Setup Pulse contact
PLS = (STEP <> LASTSTEP)
LASTSTEP = STEP

;Check if Recirculation bag needs a destination
;IF ((Bag[107].Cat > 0) AND (Bag[107].Dst = 0) AND (D[1005] > 0) AND (D[1005] <= 6) AND (D[1006] > 0)) THEN
;	Bag[107].Dst 	= D[1005]
;	D[1006] 		= (D[1006] - 1)
;ENDIF

;Step 0 - Disabled
IF (STEP = 0) THEN
	;Disabled
ENDIF

;Step 1 - Reset Ongoing Points
TON_10ms((STEP = 1),300,ResetPoints,ResetPointsET)
IF (STEP = 1) THEN
	Dest  	= 0
	Buff 	= 0
	O_Reset = NOT ResetPoints
	IF (ResetPoints AND OnGoingEnable) THEN
		D[904] = 2
	ENDIF
ENDIF

;Set Max Buffers to search
MaxBuffers = 1

;Bag Settles at each buffer
;TON_10ms(I_BagatBuffer[1],300,SettledBuffer[1],SettledBufferET[1])
SettledBuffer[1] = I_BagatBuffer[1] ;SVC1
;TON_10ms(I_BagatBuffer[2],300,SettledBuffer[2],SettledBufferET[2])

BufferBagNum[1]		= 222
;BufferBagNum[2]	= 250

;Step 2 - Search for a valid Bag at one of the buffers
IF (STEP = 2) THEN

	Buff 	= 0
	Dest 	= 0

	IF OnGoingEnable THEN

		Alarm[4].Name 	= almNoAlarm
		Alarm[4].Time	= 2000

		LOOP Bfr = 1 TO MaxBuffers DO

			;Set Test Value for Monitoring
			IF TestBuffer > 0 THEN
				Buffer = TestBuffer
			ELSE
				Buffer = Bfr
			ENDIF

			BufferBag		= BufferBagNum[Buffer]
			BufferSettled 	= SettledBuffer[Buffer]
			BufferCat 		= Bag[BufferBag].Cat
			BufferDst 		= Bag[BufferBag].Dst

			DestValid = ((BufferDst >= 1) AND (BufferDst <= Std.MaxLines))

			IF (BufferSettled AND (BufferCat > 0) AND DestValid AND (Bag[224].Cat = 0)) THEN
				n = BufferDst
				IF ((Line[n].Space > 0) AND Line[n].Clear) THEN
					Dest = n
					Buff = Buffer
					;IF (Buffer = 1) THEN
						D[904] 	= 3
					;ELSE
					;	D[904]  = 4
					;ENDIF
				ELSE
					Alarm[4].Name 	= almDestinationNotValid
					Alarm[4].Bag	= BufferBag
				ENDIF
			ENDIF

			;Buffer Alarms
			;IF (BufferCat > 0) AND NOT BufferSettled THEN
			;	Alarm[4].Name 	= almBagNotAtProx
			;	Alarm[4].Bag	= BufferBag
			;ELSE IF (BufferCat = 0) AND BufferSettled THEN
			;	Alarm[4].Name 	= almBagNotShownOnScreen
			;	Alarm[4].Bag	= BufferBag
			;ENDIF

		ENDLOOP

	ENDIF

ENDIF

;Clear Line Selections
LOOP n = 1 TO Std.MaxLines DO
	LineSelect[n] = FALSE
ENDLOOP

;Step 3 - Enable VC1 to Release a bag
IF (STEP = 3) THEN
	Enable.SPN[1] = TRUE

	IF PLS THEN
		C[Dest] = 0
	ENDIF

	LineSelect[Dest] = TRUE
	IF NOT Request.SVC[1] THEN
		D[904] = 4
	ENDIF
ENDIF

;Step 4 - Select line / open buffer stop
IF (STEP = 4) THEN

	LineSelect[Dest] 	= TRUE
	O_OpenSelect[Buff] 	= TRUE

	IF PLS THEN
		;C[Dest] = 0
		IF (Bag[224].Cat = 0) AND (Bag[BufferBagNum[Buff]].Cat > 0) THEN
			Bag[224]				 	= Bag[BufferBagNum[Buff]]
			Bag[BufferBagNum[Buff]]	 	= Bag[0]
		ENDIF
	ENDIF

	;Bag arrived on selected line
	IF Line[Dest].Trip THEN
		D[498] 						= Bag[224].Cus	;Set Customer for Customer FIFO
		Bag[224].Dst 				= 0 		    ;Clear Destination
		Bag[Line[Dest].LastBag] 	= Bag[224]
		Bag[224] 					= Bag[0]
		D[904] 						= 1
	ENDIF

	Alarm[4].Name = almBagNotArrived

ENDIF

;Alarms
TimerAlarm.IN = NOT PLS AND (Alarm[4].Name > 0) AND (AlarmOld = Alarm[4].Name)
TimerAlarm.PT = Alarm[4].Time
TimerAlarm FUB TON_10ms()
Alarm[4].On = TimerAlarm.Q
Alarm[4].ET = TimerAlarm.ET

AlarmOld = Alarm[4].Name ;Need to ensure alarm changes as may be multiple alarms on step 2

;Outputs
Y[4].Y01 = LineSelect[1] OR LineSelect[2]
Y[4].Y02 = LineSelect[3]
Y[4].Y03 = LineSelect[3]
Y[4].Y04 = LineSelect[4]
Y[4].Y05 = LineSelect[5]
Y[4].Y06 = LineSelect[6]
Y[4].Y07 = LineSelect[7]
Y[4].Y08 = LineSelect[8]
Y[4].Y09 = LineSelect[9]
Y[4].Y10 = LineSelect[10]
Y[4].Y11 = LineSelect[11]
Y[4].Y12 = LineSelect[12]
Y[4].Y13 = LineSelect[13]
Y[4].Y14 = LineSelect[14] OR O_Reset

Y[3].Y15 = LineSelect[1]
Y[3].Y14 = LineSelect[2]

END_PROGRAM
```

### Program Logical/ExportsFromOriginal/5_spf1 (IEC, version 1.00.0) - * Soiled Offgoing Transfer Lines 1 - 14

#### 5_spf1Cyclic.ab
```automation-basic
PROGRAM _CYCLIC
	(* cyclic program *)

;----------------------------------------
;Sequence 5 - SPF1 Offgoing Points D[905]
;----------------------------------------
;Inputs
;------

OffGoingEnable 		= ((D[15] > 0) AND NOT Std.HaltSys)

I_BagPassedSVC2     = X[4].X15

I_BagReleased 		= X[5].X01

I_SDCBagAtBuffer[1] = X[6].X01 	;Use for single bag buffer
I_SDCBagAtBuffer[2] = FALSE 	;X[6].X13 ;Use for single bag buffer

O_SDCBufferOpen[1]  = Y[6].Y01 OR X[6].X01 	;Use for single bag buffer
O_SDCBufferOpen[2]  = FALSE 	;Y[6].Y16 ;Use for single bag buffer

I_ApproachBrush		= X[5].X16
O_CloseBrush		= FALSE

I_BagAtStop[1] 		= X[9].X01;(Bag[Line[1].FirstBag].Cat > 0);X[5].X01
I_BagAtStop[2] 		= X[9].X02;(Bag[Line[2].FirstBag].Cat > 0);X[5].X02
I_BagAtStop[3] 		= X[9].X03;(Bag[Line[3].FirstBag].Cat > 0);X[5].X03
I_BagAtStop[4] 		= X[9].X04;(Bag[Line[4].FirstBag].Cat > 0);X[5].X04
I_BagAtStop[5] 		= X[9].X05;(Bag[Line[5].FirstBag].Cat > 0);X[5].X05
I_BagAtStop[6] 		= X[9].X06;(Bag[Line[6].FirstBag].Cat > 0);X[5].X06
I_BagAtStop[7] 		= X[9].X07;(Bag[Line[7].FirstBag].Cat > 0);X[5].X07
I_BagAtStop[8] 		= X[9].X08;(Bag[Line[8].FirstBag].Cat > 0);X[5].X08
I_BagAtStop[9] 		= X[9].X09;(Bag[Line[9].FirstBag].Cat > 0);X[5].X09
I_BagAtStop[10] 	= X[9].X10;(Bag[Line[10].FirstBag].Cat > 0);X[5].X10
I_BagAtStop[11] 	= X[9].X11;(Bag[Line[11].FirstBag].Cat > 0);X[5].X11
I_BagAtStop[12] 	= X[9].X12;(Bag[Line[12].FirstBag].Cat > 0);X[5].X12
I_BagAtStop[13] 	= X[9].X13;(Bag[Line[13].FirstBag].Cat > 0);X[5].X13
I_BagAtStop[14] 	= X[9].X14;(Bag[Line[14].FirstBag].Cat > 0);X[5].X14

O_Reset 			= FALSE
Enable.SVC[2]       = FALSE

;Buffer line configuration
;-------------------------
MaxBuffers			= 2

BufferBag[1]		= 284 ;Last buffer bag number
BufferBag[2]		= 274 ;Last buffer bag number

;Banbury Special - Empty bags from SDC2 travel on a rail close to Lines 6-14
;---------------------------------------------------------------------------
EmptyInTransit 		= (D[910] > 2)
SVC2BufferClear     = (NOT Y[6].Y01 AND NOT X[6].X01 AND Line[20].Clear AND NOT EmptyInTransit AND (Bag[230].Cat = 0))
BufferClear[1] 		= ((Line[21].Space > 0) AND NOT EmptyInTransit AND (D[21] > 0) AND (Bag[BufferBag[1]].Cat = 0))
BufferClear[2]		= ((Line[22].Space > 0) AND NOT EmptyInTransit AND (D[22] > 0) AND (Bag[BufferBag[2]].Cat = 0))
BufferClear[3]      =  (NOT X[6].X01 AND NOT Y[6].Y01  AND (Bag[230].Cat = 0) and (Bag[263].Cat = 0) and (Bag[252].Cat = 0) AND (D[916] = 2) AND NOT EmptyInTransit)

EnableSDC2Empty 	= (D[905] = 2)

;Alternating between SDC1 and SDC3
EnableSDC1Search = FALSE
EnableSDC3Search = FALSE
IF (BufferClear[1] AND BufferClear[2]) THEN
	Alternator = Alternator + 1
	IF (Alternator > 2) THEN
		Alternator = 1
	ENDIF
	IF Alternator = 1 THEN
		EnableSDC1Search = TRUE
	ELSE
		EnableSDC3Search = TRUE
	ENDIF
ENDIF

Uld[1].SDCReady 	= (BufferClear[1] AND SVC2BufferClear ) ;Passed to unloading search
Uld[2].SDCReady 	= (BufferClear[2] AND SVC2BufferClear );Passed to unloading search
Uld[3].SDCReady		= (BufferClear[3] AND SVC2BufferClear );Passed to unloading search
Uld[4].SDCReady 	= FALSE

Alarm[5].Name 		= 0
Alarm[5].Bag		= 225
Alarm[5].Beacon		= TRUE
Alarm[5].Extra		= 0
Alarm[5].Time		= 3000

;Setup Sequence
;--------------
STEP = D[905]
;Setup Pulse contact
PLS = (STEP <> LASTSTEP)
LASTSTEP = STEP

;Sequence Steps
;--------------
IF (STEP = 0) THEN
	;Disabled
ENDIF

;Step 1 - Reset Points
TON_10ms((STEP = 1),300,ResetPoints,ResetPointsET)
IF (STEP = 1) THEN
	O_Reset 	= TRUE
	FoundLine 	= 0
	Destination = 0
	;IF (ResetPoints AND OffGoingEnable) THEN
	IF (ResetPoints AND OffGoingEnable AND NOT I_BagReleased) THEN
		D[905] = 2
	ENDIF
ENDIF

;Bags on storage line timers
R_TRIG(Std.Clock100ms,IncSettle)
AlarmBagNotProx 	= FALSE
AlarmBagNotProxLine = 0

LOOP n = 1 TO Std.MaxLines DO

	LineSettle[n]  = (I_BagAtStop[n] AND (Bag[Line[n].FirstBag].Cat > 0))
	IF IncSettle AND LineSettle[n] AND (BagSettledTime[n] < $FFFF) THEN
		BagSettledTime[n] = BagSettledTime[n] + 1
	ELSE IF NOT LineSettle[n] THEN
		BagSettledTime[n] = 0
		;If Bag has destiantion and not at stop then alarm
		IF (STEP = 2) AND (Bag[Line[n].FirstBag].Dst > 0) THEN
			Alarm[5].Name	= almBagNotAtProx
			Alarm[5].Bag	= Line[n].FirstBag
			Alarm[5].Extra 	= n
		ENDIF
	ENDIF

ENDLOOP

;Buffer trip not correct alarms
LOOP n = 1 TO MaxBuffers DO
	IF (STEP = 2) AND BufferClear[n] AND NOT Uld[n].SDCReady THEN
		Alarm[5].Name 	= almSwitchFault
		Alarm[5].Bag	= BufferBag[n]
	ENDIF
ENDLOOP

;Search for the bag with a valid destination that has been waiting the longest
IF STEP = 2 THEN

	FoundLine 	= 0
	Destination = 0
	BestTime 	= 0
	SettleTime = 30 ;3 seconds

	LOOP n = 1 TO Std.MaxLines DO

		IF (BagSettledTime[n] > SettleTime) THEN
			SearchDest = Bag[Line[n].FirstBag].Dst

			SDC1_Valid  = ((SearchDest = 21) AND Uld[1].SDCReady AND (Line[21].SpaceBIT > 0))
			SDC2_Valid 	= ((SearchDest = 22) AND Uld[2].SDCReady AND (Line[22].SpaceBIT > 0))
			SDC3_Valid 	= ((SearchDest = 23) AND Uld[3].SDCReady )
			SDC4_Valid 	= ((SearchDest = 24) AND Uld[4].SDCReady)

			IF (SDC1_Valid OR SDC2_Valid OR SDC3_Valid OR SDC4_Valid) THEN
				FoundLine 	= n
				Destination = SearchDest
				BestTime 	= BagSettledTime[n]
			ENDIF
		ENDIF

	ENDLOOP

	IF ((FoundLine > 0) AND OffGoingEnable AND (Bag[225].Cat = 0) AND SVC2BufferClear AND NOT EmptyInTransit ) THEN
		D[905] = 3
	ENDIF

ENDIF

;Step 3 - Select Line / Open Stop, Until Bag at correct destination
;Clear Line Selections
LOOP n = 1 TO Std.MaxLines DO
	LineSelect[n] = FALSE
	Indication[n] = FALSE
ENDLOOP

IF (STEP = 3) THEN

	IF PLS THEN
		C[20] = 0
	ENDIF

	IF PLS  AND (Bag[225].Cat = 0) AND (Bag[Line[FoundLine].FirstBag].Cat > 0)THEN
		Bag[225] 						= Bag[Line[FoundLine].FirstBag]
		Bag[Line[FoundLine].FirstBag] 	= Bag[0]
	ENDIF

	IF I_BagReleased THEN
		CloseStop = TRUE
	ENDIF

	;Select Line - Wait for bag to arrive
	LineSelect[FoundLine] = NOT CloseStop ;TRUE
	Indication[FoundLine] = TRUE ;Use indication as single stop and display dosen't indicate to operator where the bag is comming from

	;Select Route
	IF (Destination = 21) THEN
		Uld[1].DischargerStartLine = FoundLine ;Unloading Program

		IF ((C[20] > 0) AND NOT PLS) THEN
			IF ((Bag[225].Cat > 0) AND (Bag[230].Cat = 0))THEN

				Bag[230] 	= Bag[225]
				Bag[225] 	= Bag[0]
				D[905] 		= 1
			ENDIF
		ENDIF
		LastDest = 21
	ELSE IF (Destination = 22) THEN
		Uld[2].DischargerStartLine = FoundLine ;Unloading Program
		;IF PLS THEN
		;	C[22] = 0
		;ENDIF
		;IF Line[22].Trip THEN
		IF ((C[20] > 0) AND NOT PLS) THEN
			IF ((Bag[225].Cat > 0) AND (Bag[230].Cat = 0))THEN

				Bag[230] 	= Bag[225]
				Bag[225] 	= Bag[0]
				D[905] 		= 1
			ENDIF
		ENDIF
	ELSE IF (Destination = 23) THEN
		Uld[3].DischargerStartLine = FoundLine ;Unloading Program

		IF ((C[20] > 0) AND NOT PLS) THEN
			IF ((Bag[225].Cat > 0) AND (Bag[230].Cat = 0))THEN

				Bag[230] 	= Bag[225]
				Bag[225] 	= Bag[0]
				D[905] 		= 1
			ENDIF
		ENDIF
		LastDest = 23
	ENDIF

	Alarm[5].Name	= almBagNotReleased

ELSE
	CloseStop = FALSE
ENDIF

;SSR2 Brush speed reducer
IF ((Destination = 22) AND I_ApproachBrush) THEN
	CloseBrush = TRUE
ENDIF
TON_10ms(CloseBrush,500,ResetBrush,ResetBrushET)
IF ResetBrush THEN
	CloseBrush = FALSE
ENDIF
O_CloseBrush = (CloseBrush OR EmptyInTransit) ;Brush needs closing to allow empty bags past

;Alarms
TimerAlarm.IN = NOT PLS AND (Alarm[5].Name > 0)
TimerAlarm.PT = Alarm[5].Time
TimerAlarm FUB TON_10ms()
Alarm[5].On = TimerAlarm.Q
Alarm[5].ET = TimerAlarm.ET

;Outputs
;-------
Y[5].Y15 = O_Reset

Y[5].Y01 = LineSelect[1]
Y[5].Y02 = LineSelect[2]
Y[5].Y03 = LineSelect[3]
Y[5].Y04 = LineSelect[4]
Y[5].Y05 = LineSelect[5]
Y[5].Y06 = LineSelect[6]
Y[5].Y07 = LineSelect[7]
Y[5].Y08 = LineSelect[8]
Y[5].Y09 = LineSelect[9]
Y[5].Y10 = LineSelect[10]
Y[5].Y11 = LineSelect[11]
Y[5].Y12 = LineSelect[12]
Y[5].Y13 = LineSelect[13]
Y[5].Y14 = LineSelect[14]

;Buffer line selection
Y[4].Y15 = (O_Reset OR (Destination = 21))
;Y[4].Y16 = (Destination = 22)

Y[5].Y16 = O_CloseBrush
END_PROGRAM
```

#### 5_spf1.var
```iecst
VAR RETAIN
	STEP	:UINT;
	LASTSTEP	:UINT;
	PLS	:BOOL;
	BagSettledTime	:ARRAY [0..99] OF UINT;
	Destination	:UINT;
	SettleTime	:UINT;
	BestTime	:UINT;
	LineSelect	:ARRAY [0..49] OF BOOL;
	ResetPointsET	:TIME;
	ResetPoints	:BOOL;
	n	:UINT;
	IncSettle	:BOOL;
	LineSettle	:ARRAY [0..99] OF BOOL;
	I_BagAtStop	:ARRAY [0..49] OF BOOL;
	OffGoingEnable	:BOOL;
	AlarmBagNotProx	:BOOL;
	SearchDest	:UINT;
END_VAR

VAR
	TimerAlarm	:TON_10ms;
	MaxBuffers	:UINT;
	ResetBrush	:BOOL;
	FoundLine	:UINT;
	O_Reset	:BOOL;
	O_SDCBufferOpen	:ARRAY [0..4] OF BOOL;
	I_SDCBagAtBuffer	:ARRAY [0..4] OF BOOL;
	ResetBrushET	:TIME;
	SVC2BufferClear	:BOOL;
	CloseBrush	:BOOL;
	SDC4_Valid	:BOOL;
	I_BagPassedSVC2	:BOOL;
	EnableSDC3Search	:BOOL;
	EnableSDC1Search	:BOOL;
	Alternator	:UINT;
	LastDest	:UINT;
	I_ApproachBrush	:BOOL;
	O_CloseBrush	:BOOL;
	SDC1_Valid	:BOOL;
	SDC2_Valid	:BOOL;
	SDC3_Valid	:BOOL;
	EmptyInTransit	:BOOL;
	CloseStop	:BOOL;
	I_BagReleased	:BOOL;
	BufferBag	:ARRAY [0..4] OF UINT;
	BufferClear	:ARRAY [0..4] OF BOOL;
END_VAR
```

### Program Logical/ExportsFromOriginal/6_sdc1 (IEC, version 1.00.0) - * SDC1 Machine 1 BIN/BCD

#### 6_sdc1Cyclic.ab
```automation-basic
PROGRAM _CYCLIC
	(* cyclic program *)

;Sequence 6 - Discharger 1 D[906]

;-----------------------------------------
;Revision 1.00 19/12/2005 D.J. First Issue
;-----------------------------------------

DischargerEnable 		= ((D[16] > 0) AND NOT Std.HaltSys)

I_BagAtBuffer			= X[6].X12
I_BagAtDischarger		= X[6].X02
I_OpenBag				= CAN[2].DropLoad
I_LoadDropped			= CAN[2].LoadDropped
I_BagReleased			= X[6].X05
I_BagEmpty			  	= TRUE

I_BagAtEmptyBuffer		= FALSE ;X[11].X07
O_EmptyBagBufferOpen	= FALSE ;Y[11].Y07

O_BagReady				= FALSE
O_OpenBuffer 			= FALSE
O_Steadys				= FALSE
O_Closer				= FALSE
O_OpenBag				= FALSE
O_OpenStop				= FALSE

Request.SDC[1]			= FALSE

;Alarm
Alarm[6].Name 			= almNoAlarm ;Clear sequence alarm name
Alarm[6].Bag 			= 280
Alarm[6].Beacon			= TRUE
Alarm[6].Extra			= 0
Alarm[6].Time			= 3000

;Setup Sequence
STEP = D[906]
;Setup Pulse contact
PLS = (STEP <> LASTSTEP)
LASTSTEP = STEP

;Step 0 - Disabled
IF (STEP = 0) THEN
	;Disabled
ENDIF

;Check Status - Bag settled at buffer, no bag at discharger, bag at buffer on screen and no bag at discharger on the screen
TON_10ms(I_BagAtBuffer,300,SettledAtBuffer,SettledAtBufferET)
IF (STEP = 1) THEN
	IF (DischargerEnable AND SettledAtBuffer AND NOT I_BagAtDischarger AND (Bag[281].Cat > 0) AND (Bag[280].Cat = 0) AND NOT Std.HaltSys) THEN
	;IF (DischargerEnable AND NOT I_BagAtDischarger AND (Bag[260].Cat = 0) AND NOT Std.HaltSys) THEN
		D[906] = 2
	ENDIF
	IF (Bag[280].Cat > 0) THEN
		Alarm[6].Name = almBagDataError
	ELSE IF I_BagAtDischarger THEN
		Alarm[6].Name = almSwitchFault
	ELSE IF (Bag[281].Cat > 0) AND NOT I_BagAtBuffer THEN
		Alarm[6].Name 	= almBagNotAtProx
		Alarm[6].Bag	= 281
	ELSE IF (Bag[281].Cat = 0) AND I_BagAtBuffer THEN
		Alarm[6].Name 	= almBagNotShownOnScreen
		Alarm[6].Bag	= 281
	ENDIF
ENDIF

;Wait for bag in discharger
IF (STEP = 2) THEN
	O_OpenBuffer 	= TRUE
	IF I_BagAtDischarger THEN
		D[906] = 3
	ENDIF
	Alarm[6].Name = almBagNotArrived
ENDIF

;Let bag settle in discharger
TON_10ms(((STEP = 3) AND I_BagAtDischarger),1000,SettledAtDischarger,SettledAtDischargerET)
IF (STEP = 3) THEN
	IF PLS  AND (Bag[280].Cat = 0) AND (Bag[281].Cat > 0) THEN
		Bag[280] = Bag[281]
		Bag[281] = Bag[0]
	ENDIF
	IF SettledAtDischarger THEN
		D[906] = 4
	ENDIF
	;IF ((Bag[280].Cat > 0) AND (Bag[280].Dst = 23)) THEN
	;	D[906] = 11
	;ENDIF
	Alarm[6].Name = almBagNotSettled
ENDIF

;Allow steadys to move down
TON_10ms((STEP = 4),400,SteadysDown,SteadysDownET)
IF (STEP = 4) THEN
	IF SteadysDown THEN
		D[906] = 5
	ENDIF
	IF (Bag[280].Cat = Std.MaxCats) THEN
		D[906] = 8
	ENDIF
ENDIF

;Steady cylinders on from steps 4 - 9
O_Steadys = ((STEP >= 4) AND (STEP <= 9))

;Bag opener on from step 5 - 8
O_OpenBag = ((STEP >= 6) AND (STEP <= 8))

CodeStep  = ((STEP >= 4) AND (STEP <= 5))

;Wash Codes
IF CodeStep THEN
;round up weight to give to wash machine
	Remainder = SINT(Bag[280].Wgt MOD 10)
	IF (Remainder > 4) THEN
		WgtRound = (Bag[280].Wgt + 10)
	ELSE
		WgtRound = Bag[280].Wgt
	ENDIF

	;WashCodes
	;if Below the Machine limit of 99 and no WashCode has been entered then send the Category
	;IF (Bag[260].Cat < 99) THEN
	;	WashCode = D[2000 + Bag[260].Cat]
	;	IF WashCode = 0 THEN
	;		WashCode = E[1420]
	;	ENDIF
	;ELSE IF Bag[260].Cat < Std.MaxCats THEN
	;	WashCode = D[2000 + Bag[260].Cat]
	;ELSE
	;	WashCode = 0
	;ENDIF

	CAN[2].Category 	= Bag[280].Cat
	CAN[2].Customer 	= Bag[280].Cus
	CAN[2].Weight   	= (WgtRound / 10) ;rounded up weight divide by 10
	CAN[2].DoubleLoad 	= FALSE
ELSE
	CAN[2].Category 	= 0
	CAN[2].Customer 	= 0
	CAN[2].Weight   	= 0
	CAN[2].DoubleLoad 	= FALSE
ENDIF

;Bag Ready to Washing Machine
IF (STEP = 5) THEN
	O_BagReady = TRUE
	IF I_OpenBag OR TestDischarger THEN
		D[906] = 6
	ENDIF
	;Edited destination if UT has a prob
	;IF (Bag[260].Dst = 23) THEN
	;;	D[906] = 11
	;ENDIF
ENDIF

;Set LoadDropped to False
IF (STEP <> 6) THEN
	LoadDropped = FALSE
ENDIF

;Open Bag Until LoadDropped recieved and has been open for 6 seconds
TON_10ms((STEP = 6),600,MinOpen,MinOpenET) ;ET means Elapsed Time
IF (STEP = 6) THEN

	IF I_LoadDropped OR TestDischarger THEN
	;IF I_BagEmpty THEN
		LoadDropped = TRUE
	ENDIF

	IF (LoadDropped AND MinOpen) THEN
		;Write Report
		;------------
		IF (ReportUnloading[1].Cat = 0) THEN
			ReportUnloading[1].Cat = UINT(Bag[280].Cat)	;Category
			ReportUnloading[1].Cus = Bag[280].Cus		;Customer
			ReportUnloading[1].Wgt = Bag[280].Wgt		;Weight
			ReportUnloading[1].Cnt = 0					;Count
			ReportUnloading[1].Stn = 0					;Station
			ReportUnloading[1].Mcn = 1					;Machine
		ENDIF
	ENDIF
	IF (LoadDropped AND MinOpen) THEN
		D[906] = 7
	ENDIF
	Alarm[6].Name = almLoadNotDropped
ENDIF

;Change display to empty bag
IF (STEP = 7) THEN
	IF ((NOT I_OpenBag AND NOT I_LoadDropped AND I_BagEmpty) OR TestDrop) THEN
		Bag[280].Cat 	= Std.MaxCats
		D[906] 			= 8
	ENDIF
	Alarm[6].Name = almGeneralSequence
ENDIF

;Close bag
TON_10ms((STEP = 8),700,CloserDown,CloserDownET)
IF (STEP = 8) THEN
	O_Closer = TRUE
	IF CloserDown THEN
		D[906] = 9
	ENDIF
ENDIF

;Allow closer to go back up
TON_10ms((STEP = 9),700,CloserUp,CloserUpET)
IF (STEP = 9) THEN
	IF CloserUp THEN
		D[906] = 10
	ENDIF
ENDIF

;Allow steadys to go up
TON_10ms((STEP = 10),400,SteadyUp,SteadyUpET)
IF (STEP = 10) THEN
	IF SteadyUp THEN
		D[906] = 11
	ENDIF
ENDIF

;Check for space on empty bag buffer
IF (STEP = 11) THEN
	Request.SDC[1] = TRUE
	IF Enable.SDC[1] THEN
		D[906] = 12
	ENDIF
ENDIF

;Open buffer stop - unitl bag out
IF (STEP = 12) THEN
	O_OpenStop = TRUE

	IF (Bag[280].Cat > 0) THEN
		Bag[280] = Bag[0]
	ENDIF

	IF NOT Enable.SDC[1] THEN
		D[906] = 1
	ENDIF
	Alarm[6].Name = almBagNotReleased
ENDIF

;Alarms
TimerAlarm.IN 	= NOT PLS AND (Alarm[6].Name > 0)
TimerAlarm.PT 	= Alarm[6].Time
TimerAlarm FUB TON_10ms()
Alarm[6].On 	= TimerAlarm.Q
Alarm[6].ET 	= TimerAlarm.ET

;Outputs
CAN[2].BagReady 	= O_BagReady
Y[6].Y15 			= O_OpenBuffer
Y[6].Y02 			= O_Steadys
Y[6].Y03 			= O_OpenBag
Y[6].Y04 			= O_Closer
Y[6].Y05 			= O_OpenStop
END_PROGRAM
```

#### 6_sdc1.var
```iecst
VAR RETAIN
	STEP	:UINT;
	PLS	:BOOL;
	LASTSTEP	:UINT;
	SteadyUp	:BOOL;
	CloserUpET	:TIME;
	SteadysDown	:BOOL;
	SteadysDownET	:TIME;
	LoadDropped	:BOOL;
	SteadyUpET	:TIME;
	CloserDownET	:TIME;
	SettledAtDischargerET	:TIME;
	MinOpenET	:TIME;
	SettledAtDischarger	:BOOL;
	CloserDown	:BOOL;
	MinOpen	:BOOL;
	CloserUp	:BOOL;
	SettledAtBuffer	:BOOL;
	SettledAtBufferET	:TIME;
	I_BagAtBuffer	:BOOL;
	O_OpenStop	:BOOL;
	O_OpenBag	:BOOL;
	O_Steadys	:BOOL;
	O_OpenBuffer	:BOOL;
	O_Closer	:BOOL;
	I_BagAtDischarger	:BOOL;
	I_OpenBag	:BOOL;
	I_LoadDropped	:BOOL;
	TestDrop	:BOOL;
END_VAR

VAR
	DischargerEnable	:BOOL;
	TestDischarger	:BOOL;
	I_BagEmpty	:BOOL;
	O_BagReady	:BOOL;
	I_BagReleased	:BOOL;
	O_EmptyBagBufferOpen	:BOOL;
	I_BagAtEmptyBuffer	:BOOL;
	TimerAlarm	:TON_10ms;
	CodeStep	:BOOL;
	BCD_BIN_CAT	:BCD_BIN_OUTPUT;
	BCD_BIN_CUS	:BCD_BIN_OUTPUT;
	BCD_BIN_WGT	:BCD_BIN_OUTPUT;
	Remainder	:UINT;
	WgtRound	:UINT;
END_VAR
```

### Program Logical/ExportsFromOriginal/7_sdc2 (IEC, version 1.00.0) - * SDC2 Machine 2 CAN

#### 7_sdc2Cyclic.ab
```automation-basic
PROGRAM _CYCLIC
	(* cyclic program *)

;Sequence 7 - Discharger 2 D[907]

;-----------------------------------------
;Revision 1.00 19/12/2005 D.J. First Issue
;-----------------------------------------

DischargerEnable 		= ((D[17] > 0) AND NOT Std.HaltSys)

I_BagAtBuffer			= X[6].X06
I_BagAtDischarger		= X[6].X07
I_OpenBag				= CAN[1].DropLoad
I_LoadDropped			= CAN[1].LoadDropped
I_BagReleased			= X[6].X10
I_BagEmpty			  	= TRUE
I_DischargerBagEmpty    = X[6].X11

I_BagAtEmptyBuffer		= FALSE ;X[6].X13
O_EmptyBagBufferOpen	= FALSE ;Y[6].Y13

O_BagReady				= FALSE
O_OpenBuffer 			= FALSE
O_Steadys				= FALSE
O_Closer				= FALSE
O_OpenBag				= FALSE
O_OpenStop				= FALSE

Request.SDC[2] 			= FALSE

;Alarm
Alarm[7].Name 			= almNoAlarm ;Clear sequence alarm name
Alarm[7].Bag 			= 270
Alarm[7].Beacon			= TRUE
Alarm[7].Extra			= 0
Alarm[7].Time			= 3000

;Setup Sequence
STEP = D[907]
;Setup Pulse contact
PLS = (STEP <> LASTSTEP)
LASTSTEP = STEP

;Step 0 - Disabled
IF (STEP = 0) THEN
	;Disabled
ENDIF

;Check Status - Bag settled at buffer, no bag at discharger, bag at buffer on screen and no bag at discharger on the screen
TON_10ms(I_BagAtBuffer,300,SettledAtBuffer,SettledAtBufferET)
IF (STEP = 1) THEN
	IF (DischargerEnable AND SettledAtBuffer AND NOT I_BagAtDischarger AND (Bag[271].Cat > 0) AND (Bag[270].Cat = 0) AND NOT Std.HaltSys) THEN
	;IF (DischargerEnable AND NOT I_BagAtDischarger AND (Bag[270].Cat = 0) AND NOT Std.HaltSys) THEN
		D[907] = 2
	ENDIF
	IF (Bag[270].Cat > 0) THEN
		Alarm[7].Name = almBagDataError
	ELSE IF I_BagAtDischarger THEN
		Alarm[7].Name = almSwitchFault
	ELSE IF (Bag[271].Cat > 0) AND NOT I_BagAtBuffer THEN
		Alarm[7].Name 	= almBagNotAtProx
		Alarm[7].Bag	= 271
	ELSE IF (Bag[271].Cat = 0) AND I_BagAtBuffer THEN
		Alarm[7].Name 	= almBagNotShownOnScreen
		Alarm[7].Bag	= 271
	ENDIF
ENDIF

;Wait for bag in discharger
IF (STEP = 2) THEN
	O_OpenBuffer 	= TRUE
	IF I_BagAtDischarger THEN
		D[907] = 3
	ENDIF
	Alarm[7].Name = almNoAlarm ;almBagNotArrived
ENDIF

;Let bag settle in discharger
TON_10ms(((STEP = 3) AND I_BagAtDischarger),1000,SettledAtDischarger,SettledAtDischargerET)
IF (STEP = 3) THEN
	IF (Bag[270].Cat = 0) AND (Bag[271].Cat > 0) THEN
		Bag[270] = Bag[271]
		Bag[271] = Bag[0]
	ENDIF
	IF SettledAtDischarger THEN
		D[907] = 4
	ENDIF
	Alarm[7].Name = almBagNotSettled
ENDIF

;Allow steadys to move down
TON_10ms((STEP = 4),400,SteadysDown,SteadysDownET)
IF (STEP = 4) THEN
	IF SteadysDown THEN
		D[907] = 5
	ENDIF
	IF (Bag[270].Cat = Std.MaxCats) THEN
		D[907] = 8
	ENDIF
ENDIF

;Steady cylinders on from steps 4 - 9
O_Steadys = ((STEP >= 4) AND (STEP <= 9))

;Bag opener on from step 5 - 8
O_OpenBag = ((STEP >= 6) AND (STEP <= 8))

CodeStep  = ((STEP >= 4) AND (STEP <= 5))

;Wash Codes
IF CodeStep THEN

	;round up weight to give to wash machine
	Remainder = SINT(Bag[270].Wgt MOD 10)
	IF (Remainder > 4) THEN
		WgtRound = (Bag[270].Wgt + 10)
	ELSE
		WgtRound = Bag[270].Wgt
	ENDIF

	;WashCodes
	;if Below the Machine limit of 99 and no WashCode has been entered then send the Category
	;IF (Bag[260].Cat < 99) THEN
	;	WashCode = D[2000 + Bag[260].Cat]
	;	IF WashCode = 0 THEN
	;		WashCode = E[1420]
	;	ENDIF
	;ELSE IF Bag[260].Cat < Std.MaxCats THEN
	;	WashCode = D[2000 + Bag[260].Cat]
	;ELSE
	;	WashCode = 0
	;ENDIF

	CAN[1].Category 	= Bag[270].Cat
	CAN[1].Customer 	= Bag[270].Cus
	CAN[1].Weight   	= (WgtRound / 10) ;rounded up weight divide by 10
	CAN[1].DoubleLoad 	= FALSE
ELSE
	CAN[1].Category 	= 0
	CAN[1].Customer 	= 0
	CAN[1].Weight   	= 0
	CAN[1].DoubleLoad 	= FALSE
ENDIF

;Bag Ready to Washing Machine
IF (STEP = 5) THEN
	O_BagReady 		= TRUE
	CAN[1].BagReady = TRUE
	IF I_OpenBag OR TestDischarger THEN
		D[907] = 6
	ENDIF
ELSE
	CAN[1].BagReady = FALSE
ENDIF

;Set LoadDropped to False
IF (STEP <> 6) THEN
	LoadDropped = FALSE
ENDIF

;Open Bag Until LoadDropped recieved and has been open for 6 seconds
TON_10ms((STEP = 6),600,MinOpen,MinOpenET) ;ET means Elapsed Time
TON_10ms((STEP = 6) AND NOT I_DischargerBagEmpty ,100,BagEmpty,BagEmptyET)

IF (STEP = 6) THEN
		I_DischargerBagEmpty
	IF I_LoadDropped  OR TestDischarger THEN
	;IF I_BagEmpty THEN
		LoadDropped = TRUE
	ENDIF

	IF (LoadDropped AND MinOpen) THEN
		;Write Report
		;------------

	ENDIF
	IF (LoadDropped AND MinOpen AND BagEmpty) THEN
		IF (ReportUnloading[2].Cat = 0) THEN
			ReportUnloading[2].Cat = UINT(Bag[270].Cat)	;Category
			ReportUnloading[2].Cus = Bag[270].Cus		;Customer
			ReportUnloading[2].Wgt = Bag[270].Wgt		;Weight
			ReportUnloading[2].Cnt = 0					;Count
			ReportUnloading[2].Stn = 0					;Station
			ReportUnloading[2].Mcn = 2					;Machine
		ENDIF
		D[907] = 7
	ENDIF
	Alarm[7].Name = almLoadNotDropped
ENDIF

;Change display to empty bag
IF (STEP = 7) THEN
	IF ((NOT I_OpenBag AND NOT I_LoadDropped AND I_BagEmpty) OR TestDrop) THEN
		Bag[270].Cat 	= Std.MaxCats
		D[907] 			= 8
	ENDIF
	Alarm[7].Name = almGeneralSequence
ENDIF

;Close bag
TON_10ms((STEP = 8),700,CloserDown,CloserDownET)
IF (STEP = 8) THEN
	O_Closer = TRUE
	IF CloserDown THEN
		D[907] = 9
	ENDIF
ENDIF

;Allow closer to go back up
TON_10ms((STEP = 9),700,CloserUp,CloserUpET)
IF (STEP = 9) THEN
	IF CloserUp THEN
		D[907] = 10
	ENDIF
ENDIF

;Allow steadys to go up
TON_10ms((STEP = 10),400,SteadyUp,SteadyUpET)
IF (STEP = 10) THEN
	IF SteadyUp THEN
		D[907] = 11
	ENDIF
ENDIF

;Request empty bag release
IF (STEP = 11) THEN
	Request.SDC[2] = TRUE
	IF (NOT I_BagReleased AND Line[15].Clear) THEN ;AND NOT I_BagAtEmptyBuffer AND NOT O_EmptyBagBufferOpen) THEN
		D[907] = 12
	ENDIF
ENDIF

;Open buffer stop - unitl bag out
IF (STEP = 12) THEN
	O_OpenStop = TRUE
	IF PLS THEN
		C[15] = 0
	ENDIF
	Bag[270].Cat = 0
	Bag[270].Cus = 0
	Bag[270].Wgt = 0
	IF I_BagReleased THEN
		D[907] = 1
	ENDIF
	Alarm[7].Name = almBagNotReleased
ENDIF

;Alarms
TimerAlarm.IN 	= NOT PLS AND (Alarm[7].Name > 0)
TimerAlarm.PT 	= Alarm[7].Time
TimerAlarm FUB TON_10ms()
Alarm[7].On 	= TimerAlarm.Q
Alarm[7].ET 	= TimerAlarm.ET

;Outputs
;Y[6].Y16 	= O_BagReady
Y[6].Y06 	= O_OpenBuffer
Y[6].Y07 	= O_Steadys
Y[6].Y08 	= O_OpenBag
Y[6].Y09 	= O_Closer
Y[6].Y10 	= O_OpenStop
END_PROGRAM
```

#### 7_sdc2.var
```iecst
VAR RETAIN
	STEP	:UINT;
	PLS	:BOOL;
	LASTSTEP	:UINT;
	SteadyUp	:BOOL;
	CloserUpET	:TIME;
	SteadysDown	:BOOL;
	SteadysDownET	:TIME;
	LoadDropped	:BOOL;
	SteadyUpET	:TIME;
	CloserDownET	:TIME;
	SettledAtDischargerET	:TIME;
	MinOpenET	:TIME;
	SettledAtDischarger	:BOOL;
	CloserDown	:BOOL;
	MinOpen	:BOOL;
	CloserUp	:BOOL;
	SettledAtBuffer	:BOOL;
	SettledAtBufferET	:TIME;
	I_BagAtBuffer	:BOOL;
	O_OpenStop	:BOOL;
	O_OpenBag	:BOOL;
	O_Steadys	:BOOL;
	O_OpenBuffer	:BOOL;
	O_Closer	:BOOL;
	I_BagAtDischarger	:BOOL;
	I_OpenBag	:BOOL;
	I_LoadDropped	:BOOL;
	TestDrop	:BOOL;
END_VAR

VAR
	DischargerEnable	:BOOL;
	TestDischarger	:BOOL;
	I_BagEmpty	:BOOL;
	O_BagReady	:BOOL;
	WgtRound	:UINT;
	TimerAlarm	:TON_10ms;
	I_BagReleased	:BOOL;
	O_EmptyBagBufferOpen	:BOOL;
	I_BagAtEmptyBuffer	:BOOL;
	Remainder	:UINT;
	CodeStep	:BOOL;
	I_DischargerBagEmpty	:BOOL;
	BagEmpty	:BOOL;
	BagEmptyET	:TIME;
END_VAR
```

### Program Logical/ExportsFromOriginal/8_svc1 (IEC, version 1.00.0) - * SVC1 Up from SLU1 & Loading

#### 8_svc1Cyclic.ab
```automation-basic
PROGRAM _CYCLIC
	(* cyclic program *)

;--------------------------------------------
;Sequence 8 - SVC1 Vertical conveyor 1 D[908]
;--------------------------------------------

;Inputs
I_CarrAtTop				= X[3].X09
I_CarrAtMiddle			= X[3].X11
I_CarrAtBottom			= X[3].X10
I_CarrAtWeighing		= X[3].X12
I_BagOnCarr				= X[3].X13
I_BagReleased			= X[3].X14

I_UpPushButton			= X[8].X01
I_DownPushButton		= X[8].X02

I_UseAsLoading			= X[8].X03
I_NoEmptyBag			= X[8].X05
I_CollectEmpty			= X[8].X04

O_MoveCarrUp			= FALSE
O_MoveCarrDown			= FALSE
O_OpenCarrStop			= FALSE

Enable.SVC[1]			= FALSE
Request.SVC[1]			= FALSE
SVC1RequestEmpty		= FALSE

Alarm[8].Name 			= 0
Alarm[8].Bag			= 222
Alarm[8].Beacon			= TRUE
Alarm[8].Extra			= 0
Alarm[8].Time			= 3000

;Setup Sequence
STEP = D[908]
;Setup Pulse contact
PLS = (STEP <> LASTSTEP)
LASTSTEP = STEP

;Sequence
IF (STEP = 0) THEN
	;Disabled
ENDIF

;Move carriage down to middle position
IF (STEP = 1) THEN
	O_MoveCarrDown = TRUE
	IF I_CarrAtMiddle THEN
		D[908] = 2
	ENDIF
	IF NOT Std.EStop THEN
		Alarm[8].Name = almCarriageMoveFault
	ENDIF
ENDIF

;Check Status
IF (STEP = 2) THEN
	IF (NOT I_BagOnCarr AND (Bag[222].Cat = 0) AND NOT I_CarrAtTop AND NOT I_BagReleased) THEN
		D[908] = 3
	ENDIF
	IF (Bag[223].Cat > 0) THEN
		Alarm[8].Name = almBagDataError
	ELSE IF I_BagOnCarr OR I_CarrAtTop OR I_BagReleased THEN
		Alarm[8].Name = almSwitchFault
	ENDIF
ENDIF

;Check opreation mode
IF (STEP = 3) THEN
	IF I_UseAsLoading AND I_NoEmptyBag THEN
		D[908] = 10 ;Loading VC mode and no empty required
	ELSE
		D[908] = 4
	ENDIF
ENDIF

;Open Buffer stop - Enable
IF (STEP = 4) THEN
	O_OpenBuffer 	= (NOT I_BagOnCarr AND I_CarrAtMiddle)
	Enable.SVC[1] 	= (NOT I_BagOnCarr AND I_CarrAtMiddle)
	SVC1RequestEmpty = I_UseAsLoading
	IF I_BagOnCarr THEN
		D[908] = 5
	ENDIF
	;Alarm[8].Name = almBagNotArrived
ENDIF

;Let bag settle on carriage
TON_10ms(I_BagOnCarr,300,BagSettledOnCarr,BagSettledOnCarrET)
IF (STEP = 5) THEN
	;IF (Bag[223].Cat = 0) AND (Bag[222].Cat > 0) THEN
	;	Bag[223] = Bag[222]
	;	Bag[222] = Bag[0]
	;ENDIF
	IF BagSettledOnCarr THEN
		IF (I_UseAsLoading AND (Bag[222].Cat = Std.MaxCats)) THEN
			D[908] = 10
		ELSE IF (Bag[200].Wgt < 550) THEN
			D[908] = 6
		ELSE IF (Bag[200].Wgt > 550) THEN
			Alarm[8].Name = almBagOverWeight
			Alarm[8].Time			= 500
		ENDIF
	ENDIF
	IF NOT BagSettledOnCarr THEN
		Alarm[8].Name = almBagNotSettled
	ENDIF
ENDIF

;Move Carriage up to top position
IF (STEP = 6) THEN
	O_MoveCarrUp = NOT I_CarrAtTop
	IF I_CarrAtTop THEN
		D[908] = 7
	ENDIF
	IF NOT Std.EStop THEN
		Alarm[8].Name = almCarriageMoveFault
	ENDIF
ENDIF

;Request Release to Ongoing
IF (STEP = 7) THEN
	Request.SVC[1]	= TRUE
	IF Enable.SPN[1] THEN
		D[908] = 8
	ENDIF
ENDIF

;Open carriage stop let bag into buffer
IF (STEP = 8) THEN
	Request.SVC[1]	= TRUE
	O_OpenCarrStop 	= I_CarrAtTop
	IF (Bag[224].Cat = 0) AND (Bag[222].Cat > 0) THEN
		Bag[224] = Bag[222]
		Bag[222] = Bag[0]
	ENDIF
	IF I_BagReleased THEN
		D[908] = 9
	ENDIF
	IF NOT Std.EStop THEN
		Alarm[8].Name = almBagNotReleased
	ENDIF
ENDIF

;Check Middle position switch
IF (STEP = 9) THEN
	IF NOT I_CarrAtMiddle THEN
		D[908] = 1
	ENDIF
	Alarm[8].Name = almSwitchFault
ENDIF

;----------------------
;End of Normal Sequence
;----------------------

;Loading Conveyor Section
;------------------------

;Check bottom switch
IF (STEP = 10) THEN
	IF NOT I_CarrAtBottom THEN
		D[908] = 11
	ENDIF
	Alarm[8].Name = almSwitchFault
ENDIF

;Move Carriage down to loading position
IF (STEP = 11) THEN
	O_MoveCarrDown = (NOT I_CarrAtBottom AND I_DownPushButton)
	IF I_CarrAtBottom THEN
		D[908] = 12
	ENDIF
ENDIF

;Move Carriage up or down to weighing level
IF (STEP = 12) THEN
	O_MoveCarrDown 	= (NOT I_CarrAtBottom AND I_DownPushButton AND NOT I_UpPushButton)
	O_MoveCarrUp 	= (NOT I_CarrAtWeighing AND NOT I_DownPushButton AND I_UpPushButton)
	IF I_CarrAtWeighing THEN
		D[908] = 13
	ENDIF
	;Cancel Loading VC Mode
	IF NOT I_UseAsLoading AND NOT I_BagOnCarr THEN
		D[908] = 16 ;Collect empty / back to loading unit position
	ENDIF
ENDIF

;Check neither push button is pressed
IF (STEP = 13) THEN
	IF (NOT I_UpPushButton AND NOT I_DownPushButton) THEN
		D[908] = 14
	ENDIF
	Alarm[16].Name = almSwitchFault
ENDIF

;Calculate weight
SVCRaw = DINT(AI351RAW_01)
SVCRaw = (SVCRaw * 1000) ;2000
IF (SVCRaw > 0) THEN
	Bag[200].Wgt = INT(SVCRaw / 32767)
ELSE
	Bag[200].Wgt = 0
ENDIF

;Check Destination Clear and up push button pressed
Status = 0
TON_10ms(((STEP = 14) AND I_UpPushButton),50,PButton,PButtonET)
IF (STEP = 14) THEN

	IF I_CollectEmpty THEN
		IF PButton AND NOT I_BagOnCarr THEN
			D[908] = 16
		ENDIF
	ELSE IF I_DownPushButton THEN
		D[908] = 11
	ELSE
		ValidDst 	= ((Bag[200].Dst >= 0) 	AND (Bag[200].Dst <= Std.MaxLines))
		ValidCat 	= ((Bag[200].Cat > 0) 	AND (Bag[200].Cat <= Std.MaxCats ))
		ValidCus 	= ((Bag[200].Cus > 0) 	AND (Bag[200].Cus <= Std.MaxCust ))

		;Machines have different weights Lines 1-5 for Powertrans
		IF (Bag[200].Dst <= 5) THEN
			ValidWgt	= (Bag[200].Wgt < 550) ;Under 52 Kg
		ELSE
			ValidWgt	= (Bag[200].Wgt < 550) ;Under 52 Kg
		ENDIF

		;Messages on the Panel
		IF NOT ValidDst THEN
			Status = 1
		ELSE IF NOT ValidCat THEN
			Status = 2
		ELSE IF NOT ValidCus THEN
			Status = 3
		ELSE IF NOT I_BagOnCarr THEN
			Status = 5
		ELSE IF NOT ValidWgt THEN
			Status = 6
		ENDIF
		IF PButton THEN
			IF (I_BagOnCarr AND ValidCus AND ValidCat AND ValidDst AND ValidWgt AND (Enable.Search = (Std.MaxStationBanks + 1))) THEN
				Status 	= 0
				Dst 	= 0
				;Read Destination
				;IF Bag[200].Dst = 0 THEN
				;	Choice[1] = D[2200 + Bag[200].Cat]
				;	Choice[2] = D[2300 + Bag[200].Cat]
				;	Choice[3] = D[2400 + Bag[200].Cat]
				;	Choice[4] = D[2500 + Bag[200].Cat]
				;ELSE
					Choice[1] = Bag[200].Dst
					Choice[2] = 0
					Choice[3] = 0
					Choice[4] = 0
				;ENDIF
				;Check 1st to 4th Choice destinations
				LOOP n = 4 DOWNTO 1 DO
					IF (Line[Choice[n]].SpaceBIT > 0) THEN
						Dst = Choice[n]
					ENDIF
				ENDLOOP

				IF (Dst > 0) THEN

					ReportLoading[n].Cat = Bag[200].Cat	;Category
					ReportLoading[n].Cus = Bag[200].Cus	;Customer
					ReportLoading[n].Wgt = Bag[200].Wgt	;Weight
					ReportLoading[n].Cnt = 0			;Count
					ReportLoading[n].Stn = 17         	;Station
					ReportLoading[n].Mcn = 0			;Machine
					;Copy Panel values to bag and goto next step
					Bag[222] 		= Bag[200]
					Bag[222].Dst 	= USINT(Dst)

					D[908] = 15

				ELSE
					Status = 4
				ENDIF

			ELSE
				;Not Valid
				O_AlarmLamp = TRUE

			ENDIF ;Valid

		ENDIF ;PButton

	ENDIF

ELSE
	O_AlarmLamp = FALSE
ENDIF

;Show Status on SVC1 Panel
IF (Enable.Search = (Std.MaxStationBanks + 1)) THEN
	SVC1Status = Status
ENDIF

;Step 15 - Check top switch
IF (STEP = 15) THEN
	IF NOT I_CarrAtTop THEN
		D[908] = 6
	ENDIF
	Alarm[16].Name = almSwitchFault
ENDIF

;End of loading VC

;Re-position carriage
;--------------------

;Move carriage up to middle position
IF (STEP = 16) THEN
	O_MoveCarrUp = TRUE
	IF I_CarrAtMiddle THEN
		D[908] = 17
	ENDIF
	IF NOT Std.EStop THEN
		Alarm[8].Name = almCarriageMoveFault
	ENDIF
ENDIF

;Move carriage past middle position
TON_10ms(((STEP = 17) AND NOT I_CarrAtMiddle),100,PastMiddle,PastMiddleET)
IF (STEP = 17) THEN
	O_MoveCarrUp = TRUE
	IF PastMiddle THEN
		D[908] = 1
	ENDIF
	IF NOT Std.EStop THEN
		Alarm[8].Name = almCarriageMoveFault
	ENDIF
ENDIF

;Alarms
TimerAlarm.IN 	= NOT PLS AND (Alarm[8].Name > 0)
TimerAlarm.PT 	= Alarm[8].Time
TimerAlarm FUB TON_10ms()
Alarm[8].On 	= TimerAlarm.Q
Alarm[8].ET 	= TimerAlarm.ET

;PLC Outputs
;-----------
Y[2].Y01 		= (O_MoveCarrUp 	AND NOT I_CarrAtTop)
Y[2].Y02 		= (O_MoveCarrDown 	AND NOT I_CarrAtBottom)
Y[2].Y04 		= (O_OpenCarrStop 	AND I_CarrAtTop)

;Don't allow forcing of carriage movement and carriage stop
YForceDisable[2].Y01 = TRUE
YForceDisable[2].Y02 = TRUE
YForceDisable[2].Y04 = TRUE

END_PROGRAM
```

#### 8_svc1.var
```iecst
VAR RETAIN
	I_CarrAtTop	:BOOL;
	I_CarrAtBottom	:BOOL;
	STEP	:UINT;
	PLS	:BOOL;
	LASTSTEP	:UINT;
	O_MoveCarrUp	:BOOL;
	O_OpenCarrStop	:BOOL;
	O_MoveCarrDown	:BOOL;
	I_BagOnCarr	:BOOL;
END_VAR

VAR
	O_OpenBuffer	:BOOL;
	BagSettledOnCarr	:BOOL;
	BagSettledOnCarrET	:TIME;
	I_BagReleased	:BOOL;
	TimerAlarm	:TON_10ms;
	I_CarrAtMiddle	:BOOL;
	I_CarrAtWeighing	:BOOL;
	I_NoEmptyBag	:BOOL;
	I_CollectEmpty	:BOOL;
	I_UseAsLoading	:BOOL;
	I_UpPushButton	:BOOL;
	I_DownPushButton	:BOOL;
	Dst	:UINT;
	PButton	:BOOL;
	SVCRaw	:DINT;
	n	:UINT;
	ValidCus	:BOOL;
	ValidWgt	:BOOL;
	O_AlarmLamp	:BOOL;
	ValidCat	:BOOL;
	Choice	:ARRAY [0..4] OF UINT;
	PButtonET	:TIME;
	Status	:UINT;
	PastMiddleET	:TIME;
	PastMiddle	:BOOL;
END_VAR
```

### Program Logical/ExportsFromOriginal/9_sic1 (IEC, version 1.00.0) - * SIC1 Incline Conveyor 1

#### 9_sic1Cyclic.ab
```automation-basic
PROGRAM _CYCLIC
	(* cyclic program *)

;---------------------------------------------------
;Sequence 12 - SIC1 Soiled Incline Conveyor 1 D[909]
;---------------------------------------------------

;Inputs

I_BagAtBuffer			= X[8].X06
I_PaddleInPosition		= X[6].X15
I_BagInIncline			= X[6].X14

O_OpenBufferStop		= FALSE
O_RunMotor 				= FALSE

I_BagAtOutgoingBuffer	= FALSE
O_OutgoingBufferOpen	= FALSE

Enable.SIC[1]			= FALSE
O_SelectSDC1            = FALSE
O_SelectSDC2            = FALSE

Alarm[9].Name 			= 0
Alarm[9].Bag			= 287
Alarm[9].Beacon			= TRUE
Alarm[9].Extra			= 0
Alarm[9].Time			= 3000

;Setup Sequence
STEP = D[909]
;Setup Pulse contact
PLS = (STEP <> LASTSTEP)
LASTSTEP = STEP

;Sequence
;Step 0 - Disabled
IF (STEP = 0) THEN
	;Disabled
ENDIF

;Run Incline until paddle in position
IF (STEP = 1) THEN
	O_RunMotor = NOT I_PaddleInPosition
	IF I_PaddleInPosition THEN
		D[909] = 2
	ENDIF
	IF NOT Std.EStop THEN
		Alarm[9].Name = almSwitchFault
	ENDIF
ENDIF

;Wait for at buffer
TON_10ms(I_BagAtBuffer,300,BagAtBuffer,BagAtBufferET)
IF (STEP = 2) THEN
	IF (BagAtBuffer AND (Bag[240].Cat > 0) AND NOT Std.HaltSys) THEN
		D[909] = 3
	ENDIF
	IF (Bag[240].Cat > 0) AND NOT I_BagAtBuffer THEN
		Alarm[9].Name 	= almBagNotAtProx
		Alarm[9].Bag	= 240
	ELSE IF (Bag[240].Cat = 0) AND I_BagAtBuffer THEN
		Alarm[9].Name 	= almBagNotShownOnScreen
		Alarm[9].Bag	= 240
	ENDIF
ENDIF

;Open Buffer stop
IF (STEP = 3) THEN
	O_OpenBufferStop 	= TRUE
	Enable.SIC[1]		= (NOT I_BagInIncline AND (Bag[240].Cat = 0))
	IF I_BagInIncline THEN
		D[909] = 4
	ENDIF
	;;Alarm[9].Name = almBagNotArrived
ENDIF

;Let bag settle at base of incline
TON_10ms((STEP = 4),300,BagSettled,BagSettledET)
IF (STEP = 4) THEN
	IF PLS AND (Bag[241].Cat = 0) AND (Bag[240].Cat > 0)  THEN
		Bag[241] = Bag[240]
		Bag[240] = Bag[0]
	ENDIF
	IF BagSettled THEN
		D[909] = 5
	ENDIF
ENDIF

;Move Bag up incline
TON_10ms((STEP = 5),800,BagNearTop,BagNearTopET)
IF (STEP = 5) THEN
	O_RunMotor = NOT BagNearTop
	IF BagNearTop THEN
		D[909] = 6
	ENDIF
	Alarm[9].Name = almSwitchFault
ENDIF

;Check for space at the ongoing buffer
;Run motor for 0.5 seconds
TON_10ms((STEP = 6),50,RunOn,RunOnET)
IF (STEP = 6) THEN
	O_RunMotor 		= NOT RunOn
	IF NOT Std.HaltSys THEN
		IF (Bag[242].Cat = 0) AND (Bag[241].Dst > 0) THEN
			Dest = Bag[241].Dst
			IF ((Dest = 21) AND Line[21].Clear AND (Bag[284].Cat = 0))THEN
				C[21]  = 0
				D[909] = 7
			ELSE IF ((Dest = 22) AND Line[22].Clear AND (Bag[274].Cat = 0))THEN
				C[22]  = 0
				D[909] = 8
			ENDIF

		ENDIF
	ENDIF
ENDIF

;Select SDCC 1 Buffer
IF (STEP = 7) THEN
	O_RunMotor 			= TRUE
	O_SelectSDC1        = TRUE

	IF ((Bag[241].Cat > 0) AND (Bag[242].Cat = 0)) THEN
		;Bag[241].Dst = 0
		Bag[242] = Bag[241]
		Bag[241] = Bag[0]
	ENDIF

	IF PLS THEN
		C[21] = 0
	ENDIF
	IF Line[21].Trip AND NOT PLS THEN
		IF ((Bag[242].Cat > 0) AND (Bag[284].Cat = 0)) THEN
			Bag[242].Dst = 0
			Bag[284] = Bag[242]
			Bag[242] = Bag[0]
		ENDIF
		D[909] = 1
	ENDIF
	;Alarm[9].Name = almBagNotReleased
ENDIF

;Select SDCC 1 Buffer
IF (STEP = 8) THEN
	O_RunMotor 			= TRUE
	O_SelectSDC2        = TRUE
	IF ((Bag[241].Cat > 0) AND (Bag[242].Cat = 0)) THEN
		;Bag[241].Dst = 0
		Bag[242] = Bag[241]
		Bag[241] = Bag[0]
	ENDIF

	IF PLS THEN
		C[22] = 0
	ENDIF
	IF (C[22] > 0) AND NOT PLS THEN
		IF ((Bag[242].Cat > 0) AND (Bag[274].Cat = 0)) THEN
			Bag[242].Dst = 0
			Bag[274] = Bag[242]
			Bag[242] = Bag[0]
		ENDIF
		D[909] = 1
	ENDIF
	;Alarm[9].Name = almBagNotReleased
ENDIF

;Alarms
TimerAlarm.IN 	= NOT PLS AND (Alarm[9].Name > 0)
TimerAlarm.PT 	= Alarm[9].Time
TimerAlarm FUB TON_10ms()
Alarm[9].On 	= TimerAlarm.Q
Alarm[9].ET 	= TimerAlarm.ET

;Outputs
Y[8].Y06 = O_OpenBufferStop
Y[2].Y09 = O_RunMotor
Y[8].Y14 = O_SelectSDC1
Y[8].Y15 = O_SelectSDC2
END_PROGRAM
```

#### 9_sic1.var
```iecst
VAR RETAIN
	STEP	:UINT;
	PLS	:BOOL;
	LASTSTEP	:UINT;
	O_OpenBufferStop	:BOOL;
	I_BagAtBuffer	:BOOL;
	O_RunMotor	:BOOL;
	BagSettled	:BOOL;
	BagSettledET	:TIME;
	BagAtBuffer	:BOOL;
	RunOnET	:TIME;
	RunOn	:BOOL;
	BagNearTopET	:TIME;
	BagNearTop	:BOOL;
	BagAtBufferET	:UDINT;
	I_BagInIncline	:BOOL;
END_VAR

VAR
	I_BagAtOutgoingBuffer	:BOOL;
	I_PaddleInPosition	:BOOL;
	O_SelectSDC1	:BOOL;
	O_SelectSDC2	:BOOL;
	Dest	:UINT;
	O_OutgoingBufferOpen	:BOOL;
	TimerAlarm	:TON_10ms;
END_VAR
```

### Program Logical/ExportsFromOriginal/10_ebt (IEC, version 1.00.0) - * EBT Empty bag transfer from SDC2

#### 10_ebtCyclic.ab
```automation-basic
PROGRAM _CYCLIC
	(* cyclic program *)

;-----------------------------------------------------
;Sequence 10 - EBT Empty bag transfer from SDC2 D[910]
;-----------------------------------------------------

;Inputs

I_BagAtBuffer			= X[6].X13

O_OpenBufferStop		= FALSE
Enable.SDC[1]           = FALSE
O_SelectPoint           = FALSE

I_BagAtSPI1BufferStop	= X[8].X12
O_SPI1BufferStopOpen	= Y[8].Y12

Alarm[10].Name 			= 0
Alarm[10].Bag			= 266
Alarm[10].Beacon		= TRUE
Alarm[10].Extra			= 0
Alarm[10].Time			= 3000

;Setup Sequence
STEP = D[910]
;Setup Pulse contact
PLS = (STEP <> LASTSTEP)
LASTSTEP = STEP

;Sequence
;Step 0 - Disabled
IF (STEP = 0) THEN
	;Disabled
ENDIF

;Step 1 - Wait for space at SPI1 buffer
IF (STEP = 1) THEN
	IF (Line[17].Clear AND NOT I_BagAtSPI1BufferStop AND NOT O_SPI1BufferStopOpen AND NOT Std.HaltSys) THEN
		D[910] = 2
	ENDIF
ENDIF

;Step 2 - Wait for bag at SDC2 empty bag buffer and enable from offgoing
TON_10ms(I_BagAtBuffer,300,SettledAtBuffer,SettledAtBufferET)
IF (STEP = 2) THEN
	IF EnableSDC2Empty THEN
		IF (Request.SDC[1] AND EnableSDC2Empty) THEN
			D[910] = 3

		ELSE IF (SettledAtBuffer AND EnableSDC2Empty) THEN
			D[910] = 4
		ENDIF
	ENDIF
ENDIF

;Enable SDC1
IF (STEP = 3) THEN
	Enable.SDC[1] = (D[905] <= 2)
	O_SelectPoint = (D[905] <= 2)
	IF PLS THEN
		C[17] = 0
		Bag[266].Cat = 99
	ENDIF
	IF Line[17].Trip THEN
		D[910] 		= 1
		Bag[266] 	= Bag[0]
	ENDIF
	Alarm[10].Name = almBagNotArrived
ENDIF

;Step 3 - Transfer empty from SDC2
IF (STEP = 4) THEN
	O_OpenBufferStop = (D[905] <= 2)
	IF PLS THEN
		C[17] = 0
		Bag[266].Cat = 99
	ENDIF
	IF Line[17].Trip THEN
		D[910] 		= 1
		Bag[266] 	= Bag[0]
	ENDIF
	Alarm[10].Name = almBagNotArrived
ENDIF

;Alarms
TimerAlarm.IN 	= NOT PLS AND (Alarm[10].Name > 0)
TimerAlarm.PT 	= Alarm[10].Time
TimerAlarm FUB TON_10ms()
Alarm[10].On 	= TimerAlarm.Q
Alarm[10].ET 	= TimerAlarm.ET

;Outputs
Y[6].Y13 = O_OpenBufferStop
Y[8].Y02 = O_SelectPoint
END_PROGRAM
```

#### 10_ebt.var
```iecst
VAR RETAIN
	STEP	:UINT;
	PLS	:BOOL;
	LASTSTEP	:UINT;
END_VAR

VAR
	O_OpenBufferStop	:BOOL;
	SettledAtBufferET	:TIME;
	I_BagAtBuffer	:BOOL;
	SettledAtBuffer	:BOOL;
	O_SPI1BufferStopOpen	:BOOL;
	I_BagAtSPI1BufferStop	:BOOL;
	TimerAlarm	:TON_10ms;
	O_SelectPoint	:BOOL;
	RequestSDC	:Undef;	(*  Datatype changed to Undef because there was no datatype set in the Automation Studio 2.x declaration *)
END_VAR
```

### Program Logical/ExportsFromOriginal/11_spi1 (IEC, version 1.00.0) - * SPI1 Pneumatic Incline Up 1

#### 11_spi1Cyclic.ab
```automation-basic
PROGRAM _CYCLIC
	(* cyclic program *)

;Sequence 11 - Pneumatic Incline 1 D[911]

;Incline Conveyor

;-----------------------------------------
;Revision 1.00 17/01/2006 D.J. First Issue
;-----------------------------------------

TON_10ms(O_MoveDown,1000,TempDownTime,TempDownTimeET)

I_BagAtBuffer			= X[8].X12
I_BaginIncline			= X[8].X13
I_CarrAtBottom			= X[8].X14
I_CarrAtTop				= X[8].X15

O_MoveDown 				= FALSE
O_OpenBufferStop		= FALSE

Request.SPI[1]			= FALSE

Alarm[11].Name 			= 0
Alarm[11].Bag			= 10011
Alarm[11].Beacon		= TRUE

;Setup Sequence
;--------------
STEP = D[911]
;Setup Pulse contact
PLS = (STEP <> LASTSTEP)
LASTSTEP = STEP

;Allow carriage to go up to top
IF (STEP = 1) THEN
	IF I_CarrAtTop THEN
		D[911] = 2
	ENDIF
	IF NOT Std.HaltSys THEN
		Alarm[11].Name = almCarriageMoveFault
	ENDIF
ENDIF

;Check for bag at buffer
TON_10ms(I_BagAtBuffer,300,BagSettledBuffer,BagSettledBufferET)
IF (STEP = 2) THEN
	IF BagSettledBuffer THEN
		D[911] = 3
	ENDIF
ENDIF

;Open Buffer Stop on steps 3
IF (STEP >= 3) AND (STEP <= 3) THEN
	O_OpenBufferStop = TRUE
ENDIF

;Wait for bag in incline
IF (STEP = 3) THEN
	IF I_BaginIncline THEN
		D[911] = 4
	ENDIF
	Alarm[11].Name = almBagNotArrived
ENDIF

;Let bag settle at base of incline
TON_10ms(I_BaginIncline,300,BagSettled,BagSettledET)
IF (STEP = 4) THEN
	IF BagSettled THEN
		D[911] = 5
	ENDIF
	Alarm[11].Name = almBagNotSettled
ENDIF

;Move carriage down to bottom
IF (STEP = 5) THEN
	O_MoveDown = TRUE
	IF I_CarrAtBottom THEN
		D[911] = 6
	ENDIF
	Alarm[11].Name = almCarriageMoveFault
ENDIF

;Allow carriage to move up to top
IF (STEP = 6) THEN
	IF I_CarrAtTop THEN
		D[911] 	= 7
	ENDIF
	Alarm[11].Name = almCarriageMoveFault
ENDIF

;Wait for space at empty bag buffer
IF (STEP = 7) THEN
	Request.SPI[1] = TRUE
	IF Line[18].Clear AND BagSettled THEN
		D[911] 	= 8
	ENDIF
ENDIF

;Move carriage down to bottom
IF (STEP = 8) THEN
	O_MoveDown = TRUE
	IF I_CarrAtBottom THEN
		D[911] = 9
	ENDIF
	Alarm[11].Name = almCarriageMoveFault
ENDIF

;Allow carriage to move up releasing bag
IF (STEP = 9) THEN
	IF PLS THEN
		C[18] = 0
	ENDIF
	IF Line[18].Trip THEN
		D[911] = 1
	ENDIF
	Alarm[11].Name = almBagNotReleased
ENDIF

;Alarms
TON_10ms(NOT PLS AND (Alarm[11].Name > 0),3000,Alarm[11].On,Alarm[11].ET)

Y[8].Y12 = O_OpenBufferStop
Y[8].Y13 = O_MoveDown
END_PROGRAM
```

### Program Logical/ExportsFromOriginal/12_sp2 (IEC, version 1.00.0) - * SP2 Empty bags from SDC1/2

#### 12_sp2Cyclic.ab
```automation-basic
PROGRAM _CYCLIC
	(* cyclic program *)

;---------------------------------------
;Sequence 12 - SP2 Single point 2 D[912]
;---------------------------------------

;Inputs

I_BagAtBuffer[1]		= FALSE ;X[11].X07
I_BagAtBuffer[2]		= X[11].X08

O_OpenBuffer[1]			= FALSE
O_OpenBuffer[2]			= FALSE

Enable.SDC[3]			= FALSE

Alarm[12].Name 			= 0
Alarm[12].Bag			= 10012
Alarm[12].Beacon		= TRUE
Alarm[12].Extra			= 0
Alarm[12].Time			= 3000

;Setup Sequence
STEP = D[912]
;Setup Pulse contact
PLS = (STEP <> LASTSTEP)
LASTSTEP = STEP

;Sequence
;Step 0 - Disabled
IF (STEP = 0) THEN
	;Disabled
ENDIF

;Step 1 - decide where to take bag from
TON_10ms(I_BagAtBuffer[1],300,SettledBuffer[1],SettledBufferET[1])
TON_10ms(I_BagAtBuffer[2],300,SettledBuffer[2],SettledBufferET[2])
TON_10ms(Line[18].Full,2000,SDC2BufferFull,SDC2BufferFullET)
IF (STEP = 1) THEN
	IF (Line[19].Clear AND NOT Std.HaltSys) THEN
		IF (SDC2BufferFull AND SettledBuffer[2]) THEN
			D[912] = 3 ;SDC2 Proirity if SPI1 buffer full
		ELSE IF Request.SDC[3] THEN
			D[912] = 2 ;SDC3
		ELSE IF SettledBuffer[2] THEN
			D[912] = 3 ;SDC2
		ENDIF
	ENDIF
ENDIF

;Step 2 - Transfer empty from SDC3
IF (STEP = 2) THEN
	O_OpenBuffer[1]	= TRUE
	Enable.SDC[3]	= TRUE
	IF PLS THEN
		C[19] = 0
	ENDIF
	IF Line[19].Trip THEN
		D[912] = 1
	ENDIF
	Alarm[12].Name = almBagNotArrived
ENDIF

;Step 3 - Transfer empty from SPI1 empty bag buffer
IF (STEP = 3) THEN
	O_OpenBuffer[2]	= TRUE
	IF PLS THEN
		C[19] = 0
	ENDIF
	IF Line[19].Trip THEN
		D[912] = 1
	ENDIF
	Alarm[12].Name = almBagNotArrived
ENDIF

;Alarms
TimerAlarm.IN 	= NOT PLS AND (Alarm[12].Name > 0)
TimerAlarm.PT 	= Alarm[12].Time
TimerAlarm FUB TON_10ms()
Alarm[12].On 	= TimerAlarm.Q
Alarm[12].ET 	= TimerAlarm.ET

;Outputs
Y[11].Y07 = O_OpenBuffer[1]
Y[11].Y08 = O_OpenBuffer[2]
END_PROGRAM
```

#### 12_sp2.var
```iecst
VAR RETAIN
	STEP	:UINT;
	PLS	:BOOL;
	LASTSTEP	:UINT;
END_VAR

VAR
	TimerAlarm	:TON_10ms;
	I_BagAtBuffer	:ARRAY [0..2] OF BOOL;
	O_OpenBuffer	:ARRAY [0..2] OF BOOL;
	SDC2BufferFullET	:TIME;
	SDC2BufferFull	:BOOL;
	SettledBufferET	:ARRAY [0..2] OF TIME;
	SettledBuffer	:ARRAY [0..2] OF BOOL;
END_VAR
```

### Program Logical/ExportsFromOriginal/13_spc1 (IEC) - * SPC1 Empty bag down

#### 13_spc1Cyclic.ab
```automation-basic
PROGRAM _CYCLIC
	(* cyclic program *)

;----------------------------------------------
;Sequence 13 - SPC1 Pneumatic Conveyor 1 D[913]
;----------------------------------------------

;Inputs
I_CarrAtTop				= X[5].X09
I_CarrAtBottom			= X[5].X10
I_BagOnCarr				= X[5].X11
I_BagReleased			= FALSE ;X[13].X04
I_BagAtBuffer			= X[5].X12

I_BagAtLLBuff			= FALSE ;X[12].X01
O_LLBuffOpen			= FALSE ;Y[12].Y01

O_OpenBuffer			= FALSE
O_MoveCarrUp			= FALSE
O_MoveCarrDown			= FALSE
O_OpenCarrStop			= FALSE

Alarm[13].Name 			= 0
Alarm[13].Bag			= 10013
Alarm[13].Beacon		= TRUE
Alarm[13].Extra			= 0
Alarm[13].Time			= 3000

;Setup Sequence
STEP = D[913]
;Setup Pulse contact
PLS = (STEP <> LASTSTEP)
LASTSTEP = STEP

;Sequence
IF (STEP = 0) THEN
	;Disabled
ENDIF

;Move carriage up to top position
IF (STEP = 1) THEN
	O_MoveCarrUp = TRUE
	IF I_CarrAtTop THEN
		D[913] = 2
	ENDIF
	IF NOT Std.EStop THEN
		Alarm[13].Name = almCarriageMoveFault
	ENDIF
ENDIF

;Check Status
IF (STEP = 2) THEN
	IF (NOT I_BagOnCarr AND NOT I_CarrAtBottom) THEN
		D[913] = 3
	ENDIF
	IF I_BagOnCarr OR I_CarrAtBottom THEN
		Alarm[13].Name = almSwitchFault
	ENDIF
ENDIF

;Wait for bag at buffer
TON_10ms(I_BagAtBuffer,300,SettledBuffer,SettledBufferET)
IF (STEP = 3) THEN
	IF SettledBuffer AND NOT Std.HaltSys THEN
		D[913] = 4
	ENDIF
ENDIF

;Open Buffer stop - Enable
IF (STEP = 4) THEN
	O_OpenBuffer 	= (NOT I_BagOnCarr AND I_CarrAtTop)
	;Enable.SVC[4] 	= (NOT I_BagOnCarr AND I_CarrAtBottom)
	IF I_BagOnCarr THEN
		D[913] = 5
	ENDIF
	Alarm[13].Name = almBagNotArrived
ENDIF

;Let bag settle on carriage
TON_10ms(I_BagOnCarr,300,BagSettledOnCarr,BagSettledOnCarrET)
IF (STEP = 5) THEN
	IF BagSettledOnCarr THEN
		D[913] = 6
	ENDIF
	Alarm[13].Name = almBagNotSettled
ENDIF

;Move Carriage down to bottom position
IF (STEP = 6) THEN
	O_MoveCarrDown = TRUE
	IF I_CarrAtBottom THEN
		D[913] = 7
	ENDIF
	IF NOT Std.EStop THEN
		Alarm[13].Name = almCarriageMoveFault
	ENDIF
ENDIF

;Check if buffer is clear
IF (STEP = 7) THEN
	;IF (Line[33].Clear AND NOT I_BagAtLLBuff AND NOT O_LLBuffOpen AND NOT Std.HaltSysLoading) THEN
	IF Enable.SBS[1] THEN
		D[913] = 8
	ENDIF
	;IF NOT Std.HaltSys THEN
	;	IF I_BagReleased THEN
	;		Alarm[13].Name = almSwitchFault
	;	ENDIF
	;ENDIF
ENDIF

;Open carriage stop let bag into buffer
IF (STEP = 8) THEN
	O_OpenCarrStop = TRUE
	;IF PLS THEN
	;	C[33] = 0
	;ENDIF
	;IF Line[33].Trip THEN
	IF NOT Enable.SBS[1] THEN
		D[913] = 9
	ENDIF
	IF NOT Std.EStop THEN
		Alarm[13].Name = almBagNotReleased
	ENDIF
ENDIF

;Check Top position switch
IF (STEP = 9) THEN
	IF NOT I_CarrAtTop THEN
		D[913] = 1
	ENDIF
	Alarm[13].Name = almSwitchFault
ENDIF

;Alarms
TimerAlarm.IN 	= NOT PLS AND (Alarm[13].Name > 0)
TimerAlarm.PT 	= Alarm[13].Time
TimerAlarm FUB TON_10ms()
Alarm[13].On 	= TimerAlarm.Q
Alarm[13].ET 	= TimerAlarm.ET

;PLC Outputs
;-----------
Y[7].Y16 		= (O_OpenBuffer 	AND I_CarrAtTop)
Y[2].Y03 		= (O_MoveCarrUp 	AND NOT I_CarrAtTop)
Y[2].Y07 		= (O_MoveCarrDown 	AND NOT I_CarrAtBottom)
Y[2].Y12 		= (O_OpenCarrStop 	AND I_CarrAtBottom)

;Don't allow forcing of carriage movement and carriage stop
YForceDisable[7].Y16 = TRUE
YForceDisable[2].Y03 = TRUE
YForceDisable[2].Y07 = TRUE
YForceDisable[2].Y12 = TRUE

END_PROGRAM
```

### Program Logical/ExportsFromOriginal/14_bson (IEC, version 1.00.0) - * SBSN1 Bagstacker Ongoing 

#### 14_bsonCyclic.ab
```automation-basic
PROGRAM _CYCLIC
(* cyclic program *)

;----------------------------------------
;Sequence 14 - Ongoing Bag Stacker D[914]
;----------------------------------------

;Inputs
I_BagAtBuffer			= FALSE ;X[7].X01
I_OnLineA		  		= X[7].X02
I_TiltA					= X[7].X03
I_TiltB					= X[7].X04
I_Bagout				= X[7].X06

O_OpenBufferStop		= FALSE
O_SelectLineA			= FALSE
O_SelectLineB			= FALSE
O_OpenStops				= FALSE
O_TiltCylinder			= FALSE
O_OperatePusher			= FALSE

Request.SBS[1]			= FALSE

Alarm[14].Name 			= 0
Alarm[14].Bag			= 10014
Alarm[14].Beacon		= TRUE
Alarm[14].Extra			= 0
Alarm[14].Time			= 3000

;Setup Sequence
STEP = D[914]
;Setup Pulse contact
PLS = (STEP <> LASTSTEP)
LASTSTEP = STEP

;Sequence
IF (STEP = 0) THEN
	;Disabled
ENDIF

;Select Line 'A'
TON_10ms((STEP = 1),100,PointReset,PointResetET)
IF (STEP = 1) THEN
	O_SelectLineA = NOT PointReset
	SwtichesOk = (NOT I_OnLineA AND NOT I_TiltA AND NOT I_TiltB)
	IF SwtichesOk AND PointReset AND NOT Std.HaltSys THEN
		D[914] = 2
	ENDIF
	IF NOT SwtichesOk THEN
		Alarm[14].Name = almSwitchFault
	ENDIF
ENDIF

;Wait for bag at buffer
TON_10ms(I_BagAtBuffer,300,BagAtBuffer,BagAtBufferET)
IF (STEP = 2) THEN
	;IF BagAtBuffer THEN
		D[914] = 3
	;ENDIF
ENDIF

;Open buffer stop
IF (STEP = 3) THEN
	O_SelectLineA 		= TRUE
	O_OpenBufferStop 	= TRUE
	Enable.SBS[1]		= NOT I_OnLineA
	IF I_OnLineA THEN
		D[914] = 4
	ENDIF
	;Alarm[14].Name = almBagNotArrived
ENDIF

;Select Line 'B' and Wait for bag in Tilt position
TON_10ms((I_TiltA AND I_TiltB),300,BagAtTilt,BagAtTiltET)
IF (STEP = 4) THEN
	O_SelectLineB = TRUE
	IF BagAtTilt THEN
		D[914] = 5
	ENDIF
	Alarm[14].Name = almBagNotSettled
ENDIF

;Tilt down
TON_10ms((STEP = 5),500,TiltDown,TiltDownET)
TON_10ms(TiltDown,200,Pusher,PusherET)
IF (STEP = 5) THEN
	O_TiltCylinder = TRUE
	O_Pusher       = TiltDown and not Pusher
	IF TiltDown AND Pusher THEN
		D[914] = 6
	ENDIF
ENDIF

;Tilt up
TON_10ms((STEP = 6),500,TiltUp,TiltUpET)
IF (STEP = 6) THEN
	IF TiltUp THEN
		D[914] = 7
	ENDIF
ENDIF

;Check not full
TON_10ms(NOT I_Bagout,300,NotFull,NotFullET)
IF (STEP = 7) THEN
	IF NotFull THEN
		D[914] = 8
	ENDIF
ENDIF

;Open stops to release bag
IF (STEP = 8) THEN
	O_OpenStops = TRUE
	IF I_Bagout THEN
		D[914] = 1
	ENDIF
	Alarm[14].Name = almBagNotReleased
ENDIF

;Pusher Cylinder
TON_10ms((STEP = 8) AND NOT Pushed,500,O_OperatePusher,RequirePusherET)
TON_10ms(O_OperatePusher,500,Pushed,PushedET)

;Alarms
TimerAlarm.IN 	= NOT PLS AND (Alarm[14].Name > 0)
TimerAlarm.PT 	= Alarm[14].Time
TimerAlarm FUB TON_10ms()
Alarm[14].On 	= TimerAlarm.Q
Alarm[14].ET 	= TimerAlarm.ET

;Outputs
Y[7].Y01 = O_Pusher
Y[7].Y03 = O_SelectLineA
Y[7].Y04 = O_SelectLineB
Y[7].Y05 = O_TiltCylinder
Y[7].Y06 = O_OpenStops
Y[7].Y07 = O_OperatePusher
END_PROGRAM
```

#### 14_bson.var
```iecst
VAR RETAIN
	I_BagAtBuffer	:BOOL;
	I_OnLineA	:BOOL;
	I_TiltA	:BOOL;
	I_TiltB	:BOOL;
	I_Bagout	:BOOL;
	O_OpenBufferStop	:BOOL;
	O_SelectLineA	:BOOL;
	O_SelectLineB	:BOOL;
	O_OpenStops	:BOOL;
	O_TiltCylinder	:BOOL;
	O_OperatePusher	:BOOL;
	PLS	:BOOL;
	LASTSTEP	:UINT;
	STEP	:UINT;
	BagAtBufferET	:UDINT;
	BagAtBuffer	:BOOL;
	TiltDownET	:UDINT;
	TiltDown	:BOOL;
	TiltUpET	:UDINT;
	TiltUp	:BOOL;
	NotFullET	:UDINT;
	NotFull	:BOOL;
	RequirePusherET	:UDINT;
	Pushed	:BOOL;
	PushedET	:UDINT;
END_VAR

VAR
	BagAtTiltET	:TIME;
	BagAtTilt	:BOOL;
	PointReset	:BOOL;
	PointResetET	:TIME;
	TimerAlarm	:TON_10ms;
	SwtichesOk	:BOOL;
	Pusher	:BOOL;
	PusherET	:TIME;
	O_Pusher	:BOOL;
END_VAR
```

### Program Logical/ExportsFromOriginal/15_bsoff (IEC, version 1.00.0) - * SBSF1 Bagstacker Offgoing

#### 15_bsoffCyclic.ab
```automation-basic
PROGRAM _CYCLIC
  	(* cyclic program *)

;-----------------------------------------
;Sequence 15 - Offgoing Bag Stacker D[915]
;-----------------------------------------

;Inputs
I_RockSepA				= X[7].X08
I_RockSepB				= X[7].X09
I_TiltA					= X[7].X10
I_TiltB					= X[7].X11
I_OutLineA				= X[7].X12
I_OutLineB				= X[7].X13

O_OpenRockSep			= FALSE
O_LevelCylinder			= FALSE
O_OpenLineAStop			= FALSE
O_OpenLineBStop			= FALSE
O_SelectLineA			= FALSE
O_SelectLineB			= FALSE

Alarm[15].Name 			= 0
Alarm[15].Bag			= 10015
Alarm[15].Beacon		= TRUE
Alarm[15].Extra			= 0
Alarm[15].Time			= 3000

;Setup Sequecne
STEP = D[915]
;Setup Pulse contact
PLS = (STEP <> LASTSTEP)
LASTSTEP = STEP

;Sequence

;Select Line 'A'
TON_10ms((NOT I_TiltA AND NOT I_TiltB),100,LevelClear,LevelClearET)
IF (STEP = 1) THEN
	IF LevelClear AND NOT Std.HaltSys THEN
		D[915] = 2
	ENDIF
	IF NOT Std.HaltSys THEN
		Alarm[15].Name = almSwitchFault
	ENDIF
ENDIF

;Open seperators wait for leveller to be ready
TON_10ms(((STEP = 2) AND I_RockSepA AND I_RockSepB),200,SettledInSeps,SettledInSepsET)
IF (STEP = 2) THEN
	O_OpenRockSep = TRUE
	IF SettledInSeps THEN
		D[915] = 3
	ENDIF
	;Alarm[15].Name = almBagNotArrived
ENDIF

;Wait for bag to settle in leveller position
TON_10ms((I_TiltA AND I_TiltB),300,SettledLevel,SettledLevelET)
IF (STEP = 3) THEN
	IF SettledLevel THEN
		D[915] = 4
	ENDIF
	Alarm[15].Name = almBagNotSettled
ENDIF

;Move bag leveller down
TON_10ms((STEP = 4),500,LevellerDown,LevellerDownET)
IF (STEP = 4) THEN
	O_LevelCylinder = TRUE
	IF LevellerDown THEN
		D[915] = 5
	ENDIF
ENDIF

;Allow bag leveller to retract
TON_10ms((STEP = 5),500,LevellerUp,LevellerUpET)
IF (STEP = 5) THEN
	O_LevelCylinderUP = TRUE
	IF LevellerUp THEN
		D[915] = 6
	ENDIF
ENDIF

;Check room in Buffer
IF (STEP = 6) THEN
	IF NOT Std.HaltSys THEN
		IF Enable.SLU[1] THEN
			D[915] = 7
		ENDIF
	ENDIF
ENDIF

;Open stop on line 'A'
IF (STEP = 7) THEN
	O_OpenLineAStop = TRUE
	O_SelectLineA 	= TRUE
	;IF PLS THEN
	;	C[17] = 0
	;ENDIF
	IF I_OutLineA THEN
		D[915] = 8
	ENDIF
	Alarm[15].Name = almBagNotReleased
ENDIF

;Open stop on line 'B'
IF (STEP = 8) THEN
	O_OpenLineBStop = TRUE
	O_SelectLineA 	= TRUE
	IF I_OutLineB THEN
		D[915] = 9
	ENDIF
	Alarm[15].Name = almBagNotReleased
ENDIF

;Select bag stop and wait for bag out of leveller
IF (STEP = 9) THEN
	O_SelectLineB = TRUE
	IF NOT Enable.SLU[1] THEN
		D[915] = 1
	ENDIF
	Alarm[15].Name = almBagNotReleased
ENDIF

;Alarms
TimerAlarm.IN 	= NOT PLS AND (Alarm[15].Name > 0)
TimerAlarm.PT 	= Alarm[15].Time
TimerAlarm FUB TON_10ms()
Alarm[15].On 	= TimerAlarm.Q
Alarm[15].ET 	= TimerAlarm.ET

;Outputs
Y[7].Y08 = O_OpenRockSep
Y[7].Y09 = O_LevelCylinder
Y[7].Y10 = O_OpenLineAStop
Y[7].Y11 = O_OpenLineBStop
Y[7].Y12 = O_SelectLineA
Y[7].Y13 = O_SelectLineB

;SBS Offgoing Bagstacker Pressure relief
TON_10ms((NOT X[7].X15 AND NOT X[7].X16),500,Y[7].Y15,PRLineClearET[0])

;SPR1-3
TON_10ms((NOT X[11].X10 AND NOT X[11].X11),500,Y[11].Y10,PRLineClearET[1])
TON_10ms((NOT X[11].X12 AND NOT X[11].X13),500,Y[11].Y12,PRLineClearET[2])
;TON_10ms((NOT X805 AND NOT X806),500,Y805,PRLineClearET[3])
END_PROGRAM
```

#### 15_bsoff.var
```iecst
VAR RETAIN
	STEP	:UINT;
	PLS	:BOOL;
	LASTSTEP	:UINT;
	LevellerDownET	:TIME;
	O_LevelCylinder	:BOOL;
	O_SelectLineB	:BOOL;
	O_SelectLineA	:BOOL;
	I_OutLineB	:BOOL;
	LevellerDown	:BOOL;
	LevellerUp	:BOOL;
	LevellerUpET	:TIME;
	I_TiltB	:BOOL;	(* SPR1 Trolley past stop *)
	I_OutLineA	:BOOL;
	O_OpenRockSep	:BOOL;
	O_OpenLineAStop	:BOOL;
	O_OpenLineBStop	:BOOL;
	I_RockSepA	:BOOL;
	I_RockSepB	:BOOL;
	I_TiltA	:BOOL;	(* SBS1 ON Bag on stacker *)
	O_LevelCylinderUP	:BOOL;
END_VAR

VAR
	PRLineClearET	:ARRAY [0..4] OF TIME;
	SettledLevel	:BOOL;
	SettledLevelET	:TIME;
	SettledInSepsET	:TIME;
	SettledInSeps	:BOOL;
	LevelClearET	:TIME;
	LevelClear	:BOOL;
	TimerAlarm	:TON_10ms;
END_VAR
```

### Program Logical/ExportsFromOriginal/16_sdc3 (IEC) - * SDC3 Wash-extractors
